C09078=1066.897,11.709,-66.020,172.395,25.660,154.694
C09079=1066.890,11.459,-66.005,172.394,25.657,154.694
C09080=1066.884,11.211,-65.991,172.393,25.655,154.694
C09081=1066.878,10.961,-65.976,172.391,25.653,154.693
C09082=1066.872,10.712,-65.961,172.390,25.650,154.693
C09083=1066.866,10.462,-65.946,172.388,25.647,154.693
C09084=1066.860,10.213,-65.931,172.387,25.645,154.692
C09085=1066.854,9.963,-65.918,172.386,25.642,154.692
C09086=1066.848,9.713,-65.903,172.384,25.640,154.692
C09087=1066.841,9.464,-65.888,172.383,25.637,154.692
C09088=1066.835,9.215,-65.873,172.381,25.635,154.691
C09089=1066.829,8.965,-65.858,172.380,25.632,154.691
C09090=1066.823,8.716,-65.844,172.378,25.630,154.691
C09091=1066.817,8.466,-65.829,172.377,25.627,154.690
C09092=1066.812,8.216,-65.814,172.376,25.625,154.690
C09093=1066.806,7.967,-65.799,172.374,25.622,154.690
C09094=1066.799,7.717,-65.784,172.373,25.619,154.689
C09095=1066.794,7.468,-65.770,172.371,25.617,154.689
C09096=1066.788,7.218,-65.755,172.370,25.615,154.689
C09097=1066.782,6.969,-65.741,172.369,25.612,154.688
C09098=1066.775,6.719,-65.726,172.367,25.610,154.688
C09099=1066.770,6.471,-65.711,172.366,25.607,154.688
C09100=1066.764,6.220,-65.697,172.364,25.604,154.687
C09101=1066.757,5.971,-65.682,172.363,25.602,154.687
C09102=1066.751,5.722,-65.668,172.361,25.600,154.687
C09103=1066.745,5.472,-65.653,172.360,25.597,154.686
C09104=1066.740,5.222,-65.639,172.359,25.594,154.686
C09105=1066.733,4.973,-65.624,172.357,25.592,154.686
C09106=1066.727,4.724,-65.609,172.356,25.589,154.686
C09107=1066.721,4.473,-65.595,172.354,25.587,154.685
C09108=1066.716,4.225,-65.580,172.353,25.584,154.685
C09109=1066.709,3.975,-65.565,172.352,25.582,154.685
C09110=1066.704,3.725,-65.552,172.350,25.579,154.684
C09111=1066.697,3.476,-65.537,172.349,25.577,154.684
C09112=1066.691,3.227,-65.522,172.347,25.574,154.684
C09113=1066.685,2.976,-65.508,172.346,25.572,154.683
C09114=1066.680,2.727,-65.493,172.344,25.569,154.683
C09115=1066.673,2.478,-65.478,172.343,25.566,154.683
C09116=1066.668,2.228,-65.464,172.342,25.564,154.682
C09117=1066.661,1.979,-65.450,172.340,25.562,154.682
C09118=1066.656,1.729,-65.436,172.339,25.559,154.682
C09119=1066.650,1.480,-65.421,172.337,25.556,154.681
C09120=1066.644,1.230,-65.406,172.336,25.554,154.681
C09121=1066.638,0.981,-65.392,172.334,25.551,154.681
C09122=1066.632,0.731,-65.377,172.333,25.549,154.681
C09123=1066.626,0.482,-65.363,172.332,25.547,154.680
C09124=1066.620,0.232,-65.348,172.330,25.544,154.680
C09125=1066.614,-0.017,-65.334,172.329,25.541,154.680
C09126=1066.608,-0.266,-65.321,172.327,25.539,154.679
C09127=1066.602,-0.516,-65.306,172.326,25.536,154.679
C09128=1066.596,-0.766,-65.292,172.325,25.534,154.679
C09129=1066.590,-1.015,-65.277,172.323,25.531,154.678
C09130=1066.584,-1.265,-65.263,172.322,25.528,154.678
C09131=1066.578,-1.545,-65.247,172.320,25.526,154.678
C09132=1066.571,-1.824,-65.231,172.319,25.523,154.677
C09133=1066.564,-2.105,-65.214,172.318,25.520,154.677
C09134=1066.557,-2.385,-65.198,172.315,25.517,154.677
C09135=1066.552,-2.634,-65.184,172.314,25.515,154.676
C09136=1066.546,-2.884,-65.171,172.312,25.512,154.676
C09137=1066.540,-3.133,-65.156,172.311,25.509,154.676
C09138=1066.534,-3.383,-65.142,172.310,25.507,154.675
C09139=1066.528,-3.633,-65.127,172.308,25.505,154.675
C09140=1066.522,-3.882,-65.114,172.307,25.502,154.675
C09141=1066.515,-4.132,-65.099,172.305,25.500,154.675
C09142=1066.510,-4.381,-65.085,172.304,25.498,154.674
C09143=1066.504,-4.631,-65.071,172.303,25.495,154.674
C09144=1066.497,-4.880,-65.057,172.301,25.493,154.674
C09145=1066.492,-5.130,-65.043,172.300,25.490,154.673
C09146=1066.485,-5.379,-65.028,172.298,25.488,154.673
C09147=1066.479,-5.629,-65.014,172.297,25.485,154.673
C09148=1066.473,-5.879,-65.000,172.295,25.483,154.673
C09149=1066.467,-6.128,-64.986,172.294,25.480,154.672
C09150=1066.461,-6.377,-64.972,172.293,25.478,154.672
C09151=1066.455,-6.627,-64.958,172.291,25.476,154.672
C09152=1066.449,-6.876,-64.944,172.290,25.473,154.671
C09153=1066.443,-7.125,-64.930,172.288,25.471,154.671
C09154=1066.437,-7.376,-64.916,172.287,25.469,154.671
C09155=1066.430,-7.624,-64.902,172.285,25.466,154.671
C09156=1066.424,-7.875,-64.888,172.284,25.463,154.670
C09157=1066.419,-8.124,-64.874,172.282,25.461,154.670
C09158=1066.412,-8.373,-64.860,172.281,25.459,154.670
C09159=1066.406,-8.623,-64.846,172.280,25.456,154.669
C09160=1066.401,-8.873,-64.832,172.278,25.454,154.669
C09161=1066.395,-9.122,-64.819,172.277,25.452,154.669
C09162=1066.388,-9.372,-64.804,172.275,25.449,154.669
C09163=1066.383,-9.621,-64.790,172.274,25.447,154.668
C09164=1066.377,-9.871,-64.777,172.272,25.444,154.668
C09165=1066.370,-10.121,-64.762,172.271,25.442,154.668
C09166=1066.364,-10.369,-64.748,172.270,25.439,154.667
C09167=1066.358,-10.619,-64.734,172.268,25.437,154.667
C09168=1066.352,-10.869,-64.720,172.267,25.435,154.667
C09169=1066.346,-11.119,-64.707,172.265,25.432,154.667
C09170=1066.341,-11.368,-64.693,172.264,25.430,154.666
C09171=1066.334,-11.617,-64.679,172.262,25.428,154.666
C09172=1066.328,-11.867,-64.665,172.261,25.425,154.666
C09173=1066.323,-12.117,-64.651,172.260,25.422,154.665
C09174=1066.316,-12.366,-64.638,172.258,25.420,154.665
C09175=1066.310,-12.616,-64.624,172.257,25.418,154.665
C09176=1066.304,-12.865,-64.610,172.255,25.415,154.664
C09177=1066.299,-13.115,-64.596,172.254,25.413,154.664
C09178=1066.292,-13.365,-64.581,172.252,25.411,154.664
C09179=1066.286,-13.614,-64.568,172.251,25.408,154.664
C09180=1066.281,-13.864,-64.554,172.249,25.405,154.663
C09181=1066.274,-14.113,-64.541,172.248,25.403,154.663
C09182=1066.268,-14.363,-64.527,172.247,25.401,154.663
C09183=1066.263,-14.613,-64.513,172.245,25.398,154.662
C09184=1066.257,-14.862,-64.500,172.244,25.396,154.662
C09185=1066.251,-15.111,-64.486,172.242,25.394,154.662
C09186=1066.244,-15.361,-64.472,172.241,25.391,154.662
C09187=1066.238,-15.611,-64.459,172.239,25.389,154.661
C09188=1066.233,-15.860,-64.445,172.238,25.386,154.661
C09189=1066.226,-16.109,-64.431,172.236,25.384,154.661
C09190=1066.220,-16.359,-64.417,172.235,25.382,154.661
C09191=1066.214,-16.608,-64.404,172.234,25.379,154.660
C09192=1066.208,-16.858,-64.390,172.232,25.377,154.660
C09193=1066.202,-17.108,-64.376,172.231,25.375,154.660
C09194=1066.195,-17.357,-64.363,172.229,25.372,154.660
C09195=1066.189,-17.636,-64.348,172.228,25.370,154.659
C09196=1066.182,-17.914,-64.333,172.225,25.367,154.659
C09197=1066.176,-18.193,-64.318,172.224,25.364,154.659
C09198=1066.169,-18.471,-64.302,172.223,25.362,154.658
C09199=1066.162,-18.720,-64.289,172.221,25.360,154.658
C09200=1066.156,-18.970,-64.276,172.220,25.357,154.658
C09201=1066.151,-19.220,-64.262,172.218,25.355,154.658
C09202=1066.144,-19.470,-64.249,172.217,25.353,154.657
C09203=1066.138,-19.719,-64.235,172.215,25.350,154.657
C09204=1066.132,-19.968,-64.221,172.214,25.348,154.657
C09205=1066.126,-20.218,-64.208,172.213,25.346,154.656
C09206=1066.119,-20.468,-64.195,172.211,25.343,154.656
C09207=1066.114,-20.717,-64.181,172.210,25.341,154.656
C09208=1066.108,-20.966,-64.167,172.208,25.339,154.656
C09209=1066.101,-21.216,-64.154,172.207,25.337,154.656
C09210=1066.096,-21.465,-64.140,172.205,25.334,154.655
C09211=1066.090,-21.715,-64.128,172.204,25.332,154.655
C09212=1066.083,-21.965,-64.114,172.202,25.330,154.655
C09213=1066.078,-22.215,-64.100,172.201,25.327,154.654
C09214=1066.072,-22.464,-64.087,172.199,25.325,154.654
C09215=1066.065,-22.713,-64.074,172.198,25.323,154.654
C09216=1066.060,-22.963,-64.060,172.197,25.320,154.654
C09217=1066.054,-23.212,-64.047,172.195,25.318,154.653
C09218=1066.047,-23.463,-64.034,172.194,25.316,154.653
C09219=1066.042,-23.712,-64.020,172.192,25.313,154.653
C09220=1066.035,-23.962,-64.007,172.191,25.311,154.653
C09221=1066.029,-24.211,-63.993,172.189,25.309,154.652
C09222=1066.024,-24.460,-63.979,172.187,25.306,154.652
C09223=1066.018,-24.710,-63.967,172.185,25.304,154.652
C09224=1066.012,-24.960,-63.954,172.184,25.302,154.652
C09225=1066.005,-25.209,-63.940,172.182,25.299,154.651
C09226=1066.000,-25.458,-63.926,172.181,25.297,154.651
C09227=1065.993,-25.709,-63.914,172.180,25.295,154.651
C09228=1065.987,-25.958,-63.900,172.178,25.292,154.651
C09229=1065.982,-26.208,-63.886,172.177,25.290,154.650
C09230=1065.976,-26.457,-63.873,172.175,25.288,154.650
C09231=1065.970,-26.707,-63.861,172.174,25.285,154.650
C09232=1065.963,-26.956,-63.847,172.172,25.283,154.650
C09233=1065.957,-27.205,-63.834,172.171,25.281,154.649
C09234=1065.951,-27.455,-63.821,172.169,25.279,154.649
C09235=1065.946,-27.705,-63.808,172.168,25.276,154.649
C09236=1065.939,-27.955,-63.794,172.166,25.274,154.649
C09237=1065.933,-28.205,-63.781,172.165,25.272,154.648
C09238=1065.927,-28.454,-63.768,172.163,25.270,154.648
C09239=1065.921,-28.703,-63.755,172.162,25.267,154.648
C09240=1065.915,-28.953,-63.742,172.161,25.265,154.648
C09241=1065.909,-29.202,-63.729,172.159,25.263,154.647
C09242=1065.902,-29.452,-63.716,172.158,25.261,154.647
C09243=1065.896,-29.702,-63.703,172.156,25.259,154.647
C09244=1065.890,-29.951,-63.690,172.155,25.256,154.647
C09245=1065.884,-30.201,-63.677,172.153,25.254,154.646
C09246=1065.878,-30.451,-63.664,172.152,25.252,154.646
C09247=1065.871,-30.700,-63.650,172.150,25.250,154.646
C09248=1065.865,-30.950,-63.638,172.149,25.247,154.646
C09249=1065.859,-31.199,-63.625,172.147,25.246,154.646
C09250=1065.854,-31.449,-63.612,172.146,25.243,154.645
C09251=1065.848,-31.699,-63.598,172.144,25.241,154.645
C09252=1065.842,-31.948,-63.586,172.143,25.239,154.645
C09253=1065.836,-32.198,-63.572,172.141,25.237,154.645
C09254=1065.829,-32.447,-63.559,172.140,25.234,154.644
C09255=1065.824,-32.697,-63.547,172.138,25.232,154.644
C09256=1065.817,-32.946,-63.533,172.137,25.230,154.644
C09257=1065.811,-33.196,-63.521,172.135,25.228,154.644
C09258=1065.805,-33.445,-63.508,172.134,25.226,154.643
C09259=1065.798,-33.723,-63.493,172.132,25.223,154.643
C09260=1065.791,-34.001,-63.479,172.130,25.220,154.643
C09261=1065.785,-34.279,-63.464,172.129,25.218,154.643
C09262=1065.778,-34.556,-63.450,172.127,25.216,154.642
C09263=1065.772,-34.806,-63.437,172.125,25.213,154.642
C09264=1065.766,-35.056,-63.424,172.123,25.211,154.642
C09265=1065.760,-35.305,-63.411,172.122,25.209,154.642
C09266=1065.754,-35.555,-63.399,172.121,25.207,154.641
C09267=1065.748,-35.805,-63.386,172.119,25.205,154.641
C09268=1065.742,-36.054,-63.373,172.118,25.202,154.641
C09269=1065.737,-36.303,-63.361,172.116,25.200,154.641
C09270=1065.730,-36.552,-63.347,172.115,25.198,154.641
C09271=1065.724,-36.802,-63.335,172.113,25.196,154.640
C09272=1065.718,-37.051,-63.322,172.112,25.194,154.640
C09273=1065.712,-37.301,-63.309,172.110,25.192,154.640
C09274=1065.706,-37.551,-63.296,172.109,25.189,154.640
C09275=1065.700,-37.801,-63.283,172.107,25.187,154.639
C09276=1065.694,-38.050,-63.271,172.106,25.185,154.639
C09277=1065.688,-38.300,-63.258,172.104,25.183,154.639
C09278=1065.682,-38.550,-63.245,172.103,25.181,154.639
C09279=1065.676,-38.799,-63.233,172.101,25.179,154.639
C09280=1065.670,-39.049,-63.220,172.100,25.176,154.638
C09281=1065.663,-39.298,-63.207,172.098,25.175,154.638
C09282=1065.658,-39.548,-63.194,172.097,25.172,154.638
C09283=1065.652,-39.798,-63.182,172.095,25.170,154.638
C09284=1065.645,-40.047,-63.169,172.094,25.168,154.637
C09285=1065.639,-40.297,-63.157,172.092,25.166,154.637
C09286=1065.633,-40.547,-63.144,172.091,25.164,154.637
C09287=1065.627,-40.796,-63.131,172.089,25.162,154.637
C09288=1065.621,-41.046,-63.118,172.088,25.160,154.637
C09289=1065.614,-41.295,-63.106,172.086,25.158,154.637
C09290=1065.609,-41.545,-63.094,172.085,25.156,154.636
C09291=1065.603,-41.794,-63.081,172.083,25.154,154.636
C09292=1065.597,-42.044,-63.068,172.081,25.151,154.636
C09293=1065.590,-42.293,-63.056,172.079,25.149,154.636
C09294=1065.584,-42.543,-63.044,172.078,25.147,154.635
C09295=1065.578,-42.793,-63.031,172.076,25.145,154.635
C09296=1065.572,-43.042,-63.018,172.075,25.143,154.635
C09297=1065.565,-43.292,-63.006,172.073,25.141,154.635
C09298=1065.559,-43.542,-62.993,172.072,25.139,154.635
C09299=1065.554,-43.792,-62.981,172.070,25.137,154.635
C09300=1065.548,-44.042,-62.968,172.069,25.134,154.634
C09301=1065.541,-44.290,-62.956,172.067,25.133,154.634
C09302=1065.535,-44.540,-62.943,172.066,25.130,154.634
C09303=1065.529,-44.790,-62.931,172.064,25.128,154.634
C09304=1065.524,-45.040,-62.918,172.063,25.126,154.633
C09305=1065.517,-45.289,-62.906,172.061,25.124,154.633
C09306=1065.511,-45.539,-62.894,172.060,25.122,154.633
C09307=1065.505,-45.789,-62.881,172.058,25.120,154.633
C09308=1065.499,-46.037,-62.869,172.057,25.118,154.633
C09309=1065.493,-46.287,-62.856,172.055,25.116,154.632
C09310=1065.487,-46.537,-62.844,172.054,25.114,154.632
C09311=1065.481,-46.787,-62.831,172.052,25.112,154.632
C09312=1065.474,-47.036,-62.819,172.051,25.110,154.632
C09313=1065.468,-47.286,-62.807,172.049,25.108,154.632
C09314=1065.463,-47.535,-62.795,172.048,25.106,154.631
C09315=1065.456,-47.785,-62.783,172.046,25.103,154.631
C09316=1065.451,-48.035,-62.770,172.045,25.102,154.631
C09317=1065.445,-48.285,-62.758,172.043,25.100,154.631
C09318=1065.439,-48.535,-62.745,172.041,25.097,154.631
C09319=1065.433,-48.783,-62.733,172.039,25.095,154.631
C09320=1065.427,-49.033,-62.721,172.038,25.093,154.630
C09321=1065.421,-49.283,-62.708,172.036,25.091,154.630
C09322=1065.414,-49.533,-62.696,172.035,25.089,154.630
C09323=1065.407,-49.811,-62.682,172.033,25.087,154.630
C09324=1065.401,-50.089,-62.669,172.032,25.085,154.629
C09325=1065.394,-50.366,-62.655,172.029,25.083,154.629
C09326=1065.388,-50.644,-62.641,172.028,25.080,154.629
C09327=1065.381,-50.894,-62.630,172.026,25.078,154.629
C09328=1065.375,-51.144,-62.617,172.025,25.077,154.629
C09329=1065.369,-51.393,-62.605,172.023,25.074,154.629
C09330=1065.362,-51.643,-62.593,172.022,25.072,154.628
C09331=1065.356,-51.893,-62.580,172.020,25.071,154.628
C09332=1065.349,-52.142,-62.569,172.019,25.069,154.628
C09333=1065.344,-52.391,-62.556,172.017,25.067,154.628
C09334=1065.338,-52.642,-62.545,172.016,25.065,154.628
C09335=1065.331,-52.891,-62.533,172.014,25.063,154.628
C09336=1065.325,-53.141,-62.521,172.013,25.061,154.627
C09337=1065.319,-53.391,-62.509,172.011,25.059,154.627
C09338=1065.313,-53.640,-62.496,172.009,25.057,154.627
C09339=1065.307,-53.889,-62.484,172.008,25.056,154.627
C09340=1065.300,-54.139,-62.473,172.006,25.054,154.627
C09341=1065.294,-54.389,-62.460,172.005,25.052,154.627
C09342=1065.288,-54.639,-62.449,172.002,25.049,154.627
C09343=1065.282,-54.888,-62.437,172.001,25.048,154.626
C09344=1065.276,-55.138,-62.425,171.999,25.046,154.626
C09345=1065.269,-55.387,-62.413,171.998,25.044,154.626
C09346=1065.263,-55.637,-62.400,171.996,25.042,154.626
C09347=1065.257,-55.886,-62.388,171.995,25.040,154.626
C09348=1065.251,-56.136,-62.377,171.993,25.038,154.626
C09349=1065.245,-56.386,-62.365,171.992,25.036,154.625
C09350=1065.238,-56.636,-62.353,171.990,25.034,154.625
C09351=1065.232,-56.885,-62.341,171.988,25.033,154.625
C09352=1065.226,-57.135,-62.329,171.987,25.031,154.625
C09353=1065.220,-57.385,-62.317,171.985,25.029,154.625
C09354=1065.213,-57.634,-62.305,171.984,25.027,154.625
C09355=1065.208,-57.884,-62.293,171.982,25.025,154.625
C09356=1065.201,-58.133,-62.281,171.981,25.023,154.624
C09357=1065.195,-58.383,-62.270,171.979,25.021,154.624
C09358=1065.189,-58.633,-62.257,171.978,25.019,154.624
C09359=1065.183,-58.882,-62.246,171.976,25.018,154.624
C09360=1065.177,-59.132,-62.235,171.975,25.016,154.624
C09361=1065.171,-59.382,-62.222,171.973,25.014,154.624
C09362=1065.165,-59.631,-62.210,171.971,25.012,154.623
C09363=1065.158,-59.881,-62.199,171.969,25.010,154.623
C09364=1065.153,-60.131,-62.187,171.967,25.008,154.623
C09365=1065.146,-60.380,-62.175,171.966,25.006,154.623
C09366=1065.140,-60.629,-62.163,171.964,25.005,154.623
C09367=1065.134,-60.880,-62.151,171.963,25.003,154.623
C09368=1065.128,-61.129,-62.140,171.961,25.001,154.622
C09369=1065.122,-61.379,-62.128,171.960,24.999,154.622
C09370=1065.116,-61.629,-62.116,171.958,24.997,154.622
C09371=1065.110,-61.878,-62.104,171.957,24.995,154.622
C09372=1065.104,-62.128,-62.093,171.955,24.993,154.622
C09373=1065.097,-62.378,-62.081,171.953,24.991,154.622
C09374=1065.092,-62.627,-62.069,171.952,24.990,154.622
C09375=1065.085,-62.877,-62.058,171.950,24.988,154.621
C09376=1065.079,-63.126,-62.046,171.949,24.986,154.621
C09377=1065.074,-63.376,-62.034,171.947,24.984,154.621
C09378=1065.067,-63.626,-62.022,171.946,24.982,154.621
C09379=1065.061,-63.875,-62.011,171.944,24.981,154.621
C09380=1065.055,-64.125,-61.999,171.942,24.979,154.621
C09381=1065.049,-64.375,-61.987,171.941,24.977,154.621
C09382=1065.043,-64.624,-61.976,171.939,24.975,154.620
C09383=1065.036,-64.874,-61.964,171.938,24.973,154.620
C09384=1065.031,-65.123,-61.953,171.935,24.971,154.620
C09385=1065.025,-65.373,-61.941,171.934,24.970,154.620
C09386=1065.019,-65.623,-61.930,171.932,24.968,154.620
C09387=1065.012,-65.902,-61.917,171.931,24.966,154.620
C09388=1065.005,-66.182,-61.904,171.929,24.964,154.620
C09389=1064.998,-66.460,-61.890,171.928,24.962,154.620
C09390=1064.992,-66.740,-61.877,171.925,24.960,154.619
C09391=1064.986,-66.990,-61.866,171.924,24.958,154.619
C09392=1064.979,-67.239,-61.854,171.922,24.956,154.619
C09393=1064.973,-67.489,-61.843,171.920,24.955,154.619
C09394=1064.967,-67.738,-61.831,171.919,24.953,154.619
C09395=1064.961,-67.989,-61.819,171.917,24.951,154.619
C09396=1064.955,-68.238,-61.809,171.916,24.949,154.619
C09397=1064.949,-68.488,-61.797,171.914,24.948,154.618
C09398=1064.943,-68.737,-61.786,171.913,24.946,154.618
C09399=1064.937,-68.987,-61.773,171.911,24.944,154.618
C09400=1064.931,-69.237,-61.762,171.909,24.942,154.618
C09401=1064.925,-69.487,-61.751,171.908,24.940,154.618
C09402=1064.919,-69.736,-61.739,171.906,24.938,154.618
C09403=1064.913,-69.986,-61.728,171.905,24.937,154.618
C09404=1064.907,-70.235,-61.716,171.903,24.935,154.617
C09405=1064.901,-70.485,-61.705,171.902,24.933,154.617
C09406=1064.895,-70.735,-61.694,171.899,24.932,154.617
C09407=1064.889,-70.984,-61.682,171.897,24.930,154.617
C09408=1064.883,-71.234,-61.671,171.896,24.928,154.617
C09409=1064.877,-71.484,-61.659,171.894,24.926,154.617
C09410=1064.871,-71.733,-61.648,171.893,24.924,154.617
C09411=1064.866,-71.983,-61.637,171.891,24.922,154.617
C09412=1064.859,-72.233,-61.626,171.890,24.921,154.616
C09413=1064.853,-72.482,-61.614,171.888,24.919,154.616
C09414=1064.848,-72.732,-61.602,171.886,24.918,154.616
C09415=1064.842,-72.982,-61.591,171.885,24.916,154.616
C09416=1064.835,-73.231,-61.579,171.883,24.914,154.616
C09417=1064.829,-73.481,-61.568,171.882,24.912,154.616
C09418=1064.823,-73.731,-61.557,171.880,24.910,154.616
C09419=1064.817,-73.981,-61.546,171.879,24.909,154.616
C09420=1064.811,-74.229,-61.535,171.877,24.907,154.616
C09421=1064.805,-74.480,-61.523,171.875,24.906,154.615
C09422=1064.799,-74.729,-61.513,171.874,24.904,154.615
C09423=1064.793,-74.979,-61.501,171.872,24.903,154.615
C09424=1064.787,-75.228,-61.490,171.871,24.901,154.615
C09425=1064.781,-75.478,-61.478,171.869,24.899,154.615
C09426=1064.775,-75.728,-61.468,171.867,24.898,154.615
C09427=1064.768,-75.978,-61.456,171.866,24.896,154.615
C09428=1064.763,-76.228,-61.445,171.863,24.894,154.615
C09429=1064.756,-76.477,-61.434,171.862,24.892,154.615
C09430=1064.750,-76.727,-61.423,171.860,24.891,154.615
C09431=1064.744,-76.977,-61.411,171.858,24.889,154.614
C09432=1064.738,-77.226,-61.401,171.857,24.888,154.614
C09433=1064.732,-77.476,-61.390,171.855,24.886,154.614
C09434=1064.726,-77.726,-61.378,171.854,24.884,154.614
C09435=1064.720,-77.975,-61.367,171.852,24.883,154.614
C09436=1064.714,-78.225,-61.356,171.850,24.881,154.614
C09437=1064.707,-78.474,-61.345,171.849,24.880,154.614
C09438=1064.702,-78.724,-61.334,171.847,24.878,154.614
C09439=1064.695,-78.974,-61.323,171.846,24.876,154.614
C09440=1064.689,-79.223,-61.312,171.844,24.875,154.614
C09441=1064.683,-79.474,-61.301,171.842,24.873,154.614
C09442=1064.677,-79.723,-61.290,171.841,24.872,154.614
C09443=1064.672,-79.973,-61.279,171.839,24.870,154.613
C09444=1064.665,-80.223,-61.268,171.837,24.869,154.613
C09445=1064.659,-80.471,-61.257,171.836,24.867,154.613
C09446=1064.652,-80.721,-61.246,171.834,24.866,154.613
C09447=1064.646,-80.971,-61.235,171.833,24.864,154.613
C09448=1064.639,-81.221,-61.224,171.831,24.863,154.613
C09449=1064.634,-81.470,-61.213,171.828,24.861,154.613
C09450=1064.628,-81.720,-61.203,171.827,24.859,154.613
C09451=1064.620,-82.002,-61.190,171.825,24.858,154.613
C09452=1064.614,-82.284,-61.178,171.823,24.856,154.613
C09453=1064.606,-82.565,-61.165,171.822,24.854,154.613
C09454=1064.599,-82.846,-61.153,171.819,24.852,154.613
C09455=1064.594,-83.096,-61.142,171.818,24.851,154.613
C09456=1064.587,-83.345,-61.132,171.816,24.850,154.613
C09457=1064.581,-83.595,-61.121,171.814,24.848,154.612
C09458=1064.575,-83.845,-61.110,171.813,24.847,154.612
C09459=1064.569,-84.094,-61.100,171.811,24.845,154.612
C09460=1064.562,-84.344,-61.088,171.810,24.844,154.612
C09461=1064.557,-84.594,-61.078,171.808,24.843,154.612
C09462=1064.550,-84.844,-61.068,171.806,24.841,154.612
C09463=1064.544,-85.094,-61.057,171.805,24.839,154.612
C09464=1064.538,-85.343,-61.046,171.803,24.838,154.612
C09465=1064.531,-85.593,-61.035,171.801,24.836,154.612
C09466=1064.526,-85.843,-61.024,171.800,24.835,154.612
C09467=1064.520,-86.092,-61.014,171.798,24.833,154.612
C09468=1064.513,-86.342,-61.003,171.796,24.832,154.612
C09469=1064.507,-86.591,-60.992,171.795,24.831,154.612
C09470=1064.501,-86.841,-60.981,171.792,24.829,154.612
C09471=1064.494,-87.091,-60.970,171.790,24.828,154.612
C09472=1064.489,-87.341,-60.960,171.789,24.826,154.612
C09473=1064.483,-87.590,-60.949,171.787,24.824,154.611
C09474=1064.476,-87.840,-60.939,171.786,24.823,154.611
C09475=1064.470,-88.090,-60.928,171.784,24.822,154.611
C09476=1064.464,-88.339,-60.917,171.782,24.821,154.611
C09477=1064.458,-88.588,-60.907,171.781,24.819,154.611
C09478=1064.452,-88.839,-60.896,171.779,24.818,154.611
C09479=1064.446,-89.089,-60.885,171.777,24.816,154.611
C09480=1064.440,-89.338,-60.875,171.776,24.815,154.611
C09481=1064.434,-89.587,-60.864,171.774,24.813,154.611
C09482=1064.427,-89.837,-60.854,171.772,24.812,154.611
C09483=1064.421,-90.087,-60.843,171.771,24.811,154.611
C09484=1064.416,-90.337,-60.832,171.769,24.809,154.611
C09485=1064.409,-90.587,-60.822,171.767,24.808,154.611
C09486=1064.403,-90.836,-60.811,171.766,24.807,154.611
C09487=1064.397,-91.086,-60.801,171.764,24.805,154.611
C09488=1064.391,-91.335,-60.791,171.762,24.804,154.611
C09489=1064.385,-91.585,-60.780,171.761,24.802,154.611
C09490=1064.378,-91.835,-60.769,171.759,24.801,154.611
C09491=1064.373,-92.085,-60.759,171.757,24.800,154.611
C09492=1064.367,-92.334,-60.748,171.756,24.798,154.610
C09493=1064.361,-92.584,-60.738,171.754,24.797,154.610
C09494=1064.354,-92.834,-60.727,171.751,24.795,154.611
C09495=1064.348,-93.084,-60.717,171.750,24.794,154.610
C09496=1064.342,-93.333,-60.706,171.748,24.793,154.610
C09497=1064.337,-93.583,-60.696,171.746,24.791,154.610
C09498=1064.330,-93.832,-60.686,171.745,24.790,154.610
C09499=1064.324,-94.083,-60.674,171.743,24.789,154.610
C09500=1064.318,-94.332,-60.665,171.741,24.787,154.610
C09501=1064.312,-94.582,-60.654,171.740,24.786,154.610
C09502=1064.306,-94.831,-60.643,171.738,24.784,154.610
C09503=1064.300,-95.081,-60.633,171.736,24.783,154.610
C09504=1064.294,-95.331,-60.623,171.735,24.782,154.610
C09505=1064.288,-95.581,-60.613,171.733,24.781,154.610
C09506=1064.282,-95.831,-60.602,171.731,24.779,154.610
C09507=1064.275,-96.080,-60.591,171.730,24.778,154.610
C09508=1064.270,-96.330,-60.581,171.728,24.777,154.610
C09509=1064.264,-96.579,-60.571,171.726,24.775,154.610
C09510=1064.258,-96.829,-60.561,171.725,24.774,154.610
C09511=1064.252,-97.079,-60.550,171.723,24.773,154.610
C09512=1064.245,-97.329,-60.539,171.721,24.771,154.610
C09513=1064.240,-97.579,-60.529,171.720,24.770,154.610
C09514=1064.233,-97.828,-60.519,171.718,24.769,154.610
C09515=1064.227,-98.112,-60.508,171.715,24.767,154.610
C09516=1064.220,-98.396,-60.496,171.714,24.766,154.610
C09517=1064.213,-98.679,-60.484,171.712,24.765,154.610
C09518=1064.205,-98.963,-60.473,171.710,24.763,154.610
C09519=1064.199,-99.213,-60.462,171.708,24.762,154.610
C09520=1064.193,-99.463,-60.452,171.706,24.761,154.610
C09521=1064.187,-99.712,-60.442,171.704,24.759,154.610
C09522=1064.181,-99.962,-60.432,171.703,24.758,154.610
C09523=1064.175,-100.211,-60.422,171.701,24.757,154.610
C09524=1064.168,-100.462,-60.412,171.699,24.756,154.610
C09525=1064.162,-100.711,-60.401,171.697,24.754,154.610
C09526=1064.156,-100.961,-60.391,171.696,24.753,154.610
C09527=1064.150,-101.210,-60.381,171.694,24.752,154.610
C09528=1064.144,-101.460,-60.371,171.692,24.751,154.610
C09529=1064.138,-101.710,-60.361,171.691,24.750,154.610
C09530=1064.132,-101.959,-60.351,171.689,24.749,154.610
C09531=1064.126,-102.209,-60.341,171.687,24.748,154.610
C09532=1064.120,-102.459,-60.331,171.685,24.746,154.610
C09533=1064.113,-102.709,-60.321,171.684,24.745,154.610
C09534=1064.107,-102.959,-60.311,171.682,24.744,154.610
C09535=1064.101,-103.208,-60.300,171.680,24.743,154.610
C09536=1064.095,-103.458,-60.291,171.679,24.741,154.610
C09537=1064.089,-103.708,-60.280,171.677,24.741,154.610
C09538=1064.083,-103.957,-60.270,171.675,24.740,154.610
C09539=1064.077,-104.207,-60.261,171.673,24.738,154.610
C09540=1064.070,-104.456,-60.250,171.672,24.737,154.610
C09541=1064.065,-104.707,-60.240,171.670,24.736,154.610
C09542=1064.059,-104.956,-60.231,171.668,24.735,154.610
C09543=1064.052,-105.205,-60.220,171.667,24.734,154.610
C09544=1064.046,-105.455,-60.211,171.665,24.733,154.610
C09545=1064.041,-105.705,-60.201,171.663,24.731,154.610
C09546=1064.034,-105.955,-60.190,171.661,24.730,154.610
C09547=1064.027,-106.205,-60.180,171.660,24.729,154.610
C09548=1064.021,-106.455,-60.171,171.658,24.728,154.610
C09549=1064.016,-106.705,-60.161,171.656,24.727,154.610
C09550=1064.009,-106.954,-60.150,171.655,24.726,154.610
C09551=1064.003,-107.204,-60.141,171.653,24.725,154.610
C09552=1063.997,-107.454,-60.131,171.651,24.724,154.610
C09553=1063.991,-107.704,-60.122,171.649,24.723,154.610
C09554=1063.985,-107.953,-60.111,171.647,24.721,154.610
C09555=1063.979,-108.203,-60.101,171.645,24.720,154.610
C09556=1063.973,-108.453,-60.092,171.643,24.719,154.610
C09557=1063.966,-108.702,-60.082,171.641,24.718,154.610
C09558=1063.960,-108.952,-60.072,171.640,24.717,154.610
C09559=1063.954,-109.201,-60.062,171.638,24.716,154.610
C09560=1063.948,-109.451,-60.053,171.636,24.715,154.610
C09561=1063.941,-109.701,-60.043,171.634,24.714,154.610
C09562=1063.936,-109.951,-60.033,171.633,24.713,154.610
C09563=1063.930,-110.200,-60.023,171.631,24.712,154.610
C09564=1063.923,-110.450,-60.013,171.629,24.711,154.610
C09565=1063.917,-110.700,-60.004,171.627,24.710,154.610
C09566=1063.911,-110.950,-59.994,171.626,24.709,154.610
C09567=1063.905,-111.199,-59.984,171.624,24.708,154.610
C09568=1063.899,-111.449,-59.975,171.622,24.707,154.610
C09569=1063.893,-111.699,-59.965,171.620,24.706,154.610
C09570=1063.886,-111.948,-59.955,171.619,24.705,154.610
C09571=1063.880,-112.198,-59.945,171.617,24.704,154.611
C09572=1063.874,-112.448,-59.935,171.615,24.703,154.611
C09573=1063.868,-112.698,-59.926,171.613,24.702,154.611
C09574=1063.862,-112.948,-59.916,171.612,24.701,154.611
C09575=1063.856,-113.198,-59.907,171.610,24.700,154.611
C09576=1063.850,-113.447,-59.897,171.608,24.699,154.611
C09577=1063.844,-113.697,-59.887,171.606,24.698,154.611
C09578=1063.837,-113.947,-59.878,171.605,24.697,154.611
C09579=1063.830,-114.229,-59.867,171.603,24.696,154.611
C09580=1063.824,-114.510,-59.856,171.600,24.695,154.611
C09581=1063.817,-114.792,-59.845,171.598,24.694,154.611
C09582=1063.810,-115.074,-59.835,171.597,24.693,154.611
C09583=1063.803,-115.324,-59.825,171.595,24.692,154.611
C09584=1063.797,-115.574,-59.816,171.593,24.691,154.611
C09585=1063.791,-115.824,-59.806,171.591,24.690,154.611
C09586=1063.785,-116.074,-59.796,171.589,24.689,154.611
C09587=1063.779,-116.323,-59.787,171.588,24.688,154.611
C09588=1063.772,-116.573,-59.777,171.586,24.687,154.611
C09589=1063.766,-116.823,-59.768,171.584,24.687,154.611
C09590=1063.761,-117.072,-59.759,171.582,24.685,154.611
C09591=1063.755,-117.322,-59.749,171.581,24.685,154.612
C09592=1063.748,-117.572,-59.739,171.579,24.684,154.612
C09593=1063.742,-117.821,-59.730,171.577,24.683,154.612
C09594=1063.736,-118.071,-59.720,171.575,24.682,154.612
C09595=1063.730,-118.321,-59.711,171.573,24.681,154.612
C09596=1063.724,-118.571,-59.701,171.572,24.680,154.612
C09597=1063.718,-118.821,-59.692,171.570,24.680,154.612
C09598=1063.711,-119.070,-59.682,171.568,24.679,154.612
C09599=1063.704,-119.320,-59.673,171.566,24.678,154.612
C09600=1063.699,-119.569,-59.664,171.564,24.677,154.612
C09601=1063.693,-119.819,-59.655,171.563,24.676,154.612
C09602=1063.687,-120.069,-59.645,171.561,24.675,154.612
C09603=1063.681,-120.319,-59.636,171.559,24.674,154.612
C09604=1063.675,-120.569,-59.626,171.557,24.674,154.612
C09605=1063.668,-120.819,-59.617,171.556,24.673,154.612
C09606=1063.662,-121.068,-59.607,171.554,24.672,154.613
C09607=1063.656,-121.318,-59.598,171.552,24.671,154.613
C09608=1063.650,-121.568,-59.590,171.550,24.671,154.613
C09609=1063.644,-121.817,-59.580,171.548,24.669,154.613
C09610=1063.638,-122.067,-59.571,171.547,24.669,154.613
C09611=1063.631,-122.317,-59.561,171.545,24.668,154.613
C09612=1063.625,-122.567,-59.551,171.543,24.667,154.613
C09613=1063.619,-122.817,-59.542,171.541,24.666,154.613
C09614=1063.614,-123.066,-59.533,171.539,24.665,154.613
C09615=1063.607,-123.316,-59.524,171.537,24.665,154.613
C09616=1063.601,-123.566,-59.515,171.536,24.664,154.613
C09617=1063.595,-123.815,-59.505,171.534,24.663,154.613
C09618=1063.588,-124.065,-59.496,171.532,24.662,154.613
C09619=1063.583,-124.316,-59.487,171.530,24.662,154.614
C09620=1063.576,-124.564,-59.478,171.528,24.661,154.614
C09621=1063.570,-124.814,-59.469,171.527,24.660,154.614
C09622=1063.564,-125.064,-59.459,171.525,24.660,154.614
C09623=1063.558,-125.314,-59.450,171.523,24.659,154.614
C09624=1063.551,-125.564,-59.441,171.521,24.658,154.614
C09625=1063.546,-125.813,-59.432,171.519,24.658,154.614
C09626=1063.540,-126.063,-59.423,171.518,24.656,154.614
C09627=1063.534,-126.313,-59.414,171.516,24.656,154.614
C09628=1063.527,-126.563,-59.405,171.514,24.655,154.614
C09629=1063.520,-126.813,-59.395,171.512,24.654,154.615
C09630=1063.515,-127.062,-59.387,171.510,24.654,154.615
C09631=1063.508,-127.312,-59.378,171.508,24.653,154.615
C09632=1063.502,-127.562,-59.368,171.506,24.652,154.615
C09633=1063.496,-127.812,-59.359,171.505,24.652,154.615
C09634=1063.491,-128.061,-59.350,171.503,24.650,154.615
C09635=1063.487,-128.312,-59.339,171.501,24.649,154.615
C09636=1063.485,-128.563,-59.329,171.500,24.647,154.615
C09637=1063.484,-128.814,-59.316,171.499,24.644,154.614
C09638=1063.485,-129.064,-59.304,171.498,24.640,154.614
C09639=1063.488,-129.316,-59.290,171.497,24.636,154.613
C09640=1063.493,-129.567,-59.276,171.497,24.631,154.612
C09641=1063.498,-129.819,-59.262,171.496,24.626,154.611
C09642=1063.506,-130.069,-59.246,171.496,24.620,154.610
C09643=1063.123,-130.092,-59.431,171.448,24.772,154.643
C09644=1063.115,-129.842,-59.447,171.449,24.778,154.644
C09645=1063.110,-129.590,-59.461,171.448,24.784,154.645
C09646=1063.106,-129.339,-59.476,171.449,24.788,154.646
C09647=1063.103,-129.086,-59.490,171.450,24.792,154.647
C09648=1063.102,-128.836,-59.502,171.451,24.796,154.647
C09649=1063.102,-128.586,-59.514,171.453,24.799,154.648
C09650=1063.105,-128.335,-59.525,171.454,24.801,154.648
C09651=1063.108,-128.084,-59.535,171.456,24.803,154.648
C09652=1063.112,-127.835,-59.545,171.457,24.804,154.648
C09653=1063.119,-127.585,-59.553,171.459,24.805,154.648
C09654=1063.125,-127.335,-59.563,171.461,24.806,154.648
C09655=1063.131,-127.085,-59.572,171.463,24.806,154.648
C09656=1063.138,-126.835,-59.581,171.465,24.807,154.648
C09657=1063.144,-126.586,-59.590,171.466,24.808,154.647
C09658=1063.150,-126.336,-59.599,171.468,24.808,154.647
C09659=1063.156,-126.086,-59.609,171.470,24.809,154.647
C09660=1063.163,-125.836,-59.617,171.472,24.810,154.647
C09661=1063.169,-125.586,-59.627,171.474,24.810,154.647
C09662=1063.174,-125.337,-59.636,171.476,24.811,154.647
C09663=1063.180,-125.087,-59.645,171.478,24.812,154.647
C09664=1063.187,-124.837,-59.654,171.479,24.813,154.647
C09665=1063.193,-124.587,-59.663,171.481,24.814,154.647
C09666=1063.199,-124.338,-59.673,171.483,24.814,154.647
C09667=1063.205,-124.087,-59.682,171.485,24.815,154.646
C09668=1063.212,-123.838,-59.690,171.487,24.815,154.646
C09669=1063.218,-123.589,-59.700,171.488,24.816,154.646
C09670=1063.224,-123.339,-59.710,171.490,24.817,154.646
C09671=1063.230,-123.089,-59.719,171.492,24.818,154.646
C09672=1063.236,-122.839,-59.728,171.494,24.819,154.646
C09673=1063.242,-122.590,-59.737,171.496,24.819,154.646
C09674=1063.248,-122.340,-59.747,171.497,24.821,154.646
C09675=1063.255,-122.090,-59.756,171.499,24.821,154.646
C09676=1063.261,-121.840,-59.765,171.501,24.822,154.646
C09677=1063.267,-121.591,-59.775,171.503,24.823,154.646
C09678=1063.273,-121.340,-59.784,171.505,24.823,154.646
C09679=1063.279,-121.090,-59.793,171.506,24.824,154.646
C09680=1063.285,-120.841,-59.802,171.508,24.825,154.645
C09681=1063.291,-120.592,-59.812,171.510,24.826,154.645
C09682=1063.298,-120.342,-59.821,171.512,24.827,154.645
C09683=1063.304,-120.092,-59.831,171.514,24.828,154.645
C09684=1063.310,-119.842,-59.840,171.515,24.828,154.645
C09685=1063.316,-119.592,-59.849,171.517,24.829,154.645
C09686=1063.322,-119.342,-59.859,171.519,24.830,154.645
C09687=1063.328,-119.092,-59.868,171.521,24.831,154.645
C09688=1063.334,-118.843,-59.877,171.523,24.831,154.645
C09689=1063.340,-118.594,-59.887,171.524,24.833,154.645
C09690=1063.346,-118.344,-59.896,171.526,24.833,154.645
C09691=1063.352,-118.094,-59.906,171.528,24.835,154.645
C09692=1063.359,-117.844,-59.915,171.530,24.835,154.645
C09693=1063.365,-117.595,-59.925,171.532,24.836,154.645
C09694=1063.372,-117.345,-59.934,171.533,24.837,154.645
C09695=1063.378,-117.095,-59.944,171.535,24.838,154.644
C09696=1063.384,-116.845,-59.953,171.537,24.838,154.644
C09697=1063.390,-116.595,-59.963,171.539,24.840,154.644
C09698=1063.396,-116.346,-59.972,171.541,24.840,154.644
C09699=1063.402,-116.097,-59.982,171.542,24.842,154.644
C09700=1063.408,-115.847,-59.991,171.544,24.842,154.644
C09701=1063.414,-115.597,-60.001,171.546,24.843,154.644
C09702=1063.420,-115.347,-60.010,171.548,24.844,154.644
C09703=1063.426,-115.097,-60.020,171.549,24.845,154.644
C09704=1063.434,-114.815,-60.031,171.551,24.846,154.644
C09705=1063.440,-114.533,-60.042,171.554,24.847,154.644
C09706=1063.447,-114.251,-60.052,171.556,24.848,154.644
C09707=1063.454,-113.968,-60.063,171.557,24.849,154.644
C09708=1063.460,-113.719,-60.073,171.559,24.850,154.644
C09709=1063.467,-113.469,-60.083,171.561,24.851,154.644
C09710=1063.473,-113.220,-60.093,171.563,24.852,154.644
C09711=1063.479,-112.970,-60.102,171.564,24.853,154.644
C09712=1063.485,-112.720,-60.112,171.566,24.854,154.644
C09713=1063.491,-112.470,-60.121,171.568,24.855,154.644
C09714=1063.497,-112.220,-60.131,171.570,24.856,154.643
C09715=1063.503,-111.971,-60.140,171.572,24.857,154.643
C09716=1063.509,-111.721,-60.150,171.573,24.858,154.643
C09717=1063.515,-111.472,-60.159,171.575,24.859,154.643
C09718=1063.521,-111.222,-60.170,171.577,24.860,154.643
C09719=1063.527,-110.972,-60.180,171.579,24.861,154.643
C09720=1063.533,-110.723,-60.189,171.580,24.862,154.643
C09721=1063.540,-110.473,-60.199,171.583,24.863,154.643
C09722=1063.546,-110.223,-60.208,171.585,24.864,154.643
C09723=1063.552,-109.973,-60.218,171.586,24.865,154.643
C09724=1063.558,-109.724,-60.228,171.588,24.866,154.643
C09725=1063.565,-109.474,-60.238,171.590,24.867,154.643
C09726=1063.571,-109.224,-60.248,171.592,24.869,154.643
C09727=1063.577,-108.974,-60.258,171.594,24.869,154.643
C09728=1063.583,-108.724,-60.267,171.595,24.870,154.643
C09729=1063.589,-108.475,-60.278,171.597,24.871,154.643
C09730=1063.596,-108.225,-60.287,171.599,24.872,154.643
C09731=1063.602,-107.975,-60.297,171.600,24.874,154.643
C09732=1063.608,-107.725,-60.306,171.602,24.874,154.643
C09733=1063.614,-107.476,-60.317,171.604,24.875,154.643
C09734=1063.620,-107.226,-60.327,171.606,24.877,154.643
C09735=1063.626,-106.976,-60.336,171.607,24.878,154.643
C09736=1063.632,-106.726,-60.346,171.609,24.879,154.643
C09737=1063.639,-106.477,-60.356,171.611,24.880,154.643
C09738=1063.645,-106.227,-60.366,171.613,24.881,154.643
C09739=1063.650,-105.977,-60.376,171.614,24.882,154.643
C09740=1063.657,-105.728,-60.386,171.616,24.883,154.643
C09741=1063.663,-105.478,-60.396,171.618,24.884,154.643
C09742=1063.669,-105.228,-60.405,171.620,24.885,154.643
C09743=1063.675,-104.978,-60.416,171.621,24.887,154.643
C09744=1063.681,-104.729,-60.426,171.623,24.888,154.643
C09745=1063.687,-104.479,-60.435,171.625,24.888,154.643
C09746=1063.693,-104.229,-60.446,171.627,24.890,154.643
C09747=1063.700,-103.979,-60.456,171.628,24.891,154.643
C09748=1063.706,-103.730,-60.466,171.630,24.892,154.643
C09749=1063.712,-103.480,-60.476,171.632,24.893,154.643
C09750=1063.718,-103.230,-60.486,171.633,24.895,154.643
C09751=1063.724,-102.981,-60.496,171.635,24.895,154.643
C09752=1063.730,-102.731,-60.506,171.637,24.897,154.643
C09753=1063.736,-102.481,-60.516,171.639,24.898,154.643
C09754=1063.742,-102.232,-60.527,171.640,24.899,154.643
C09755=1063.749,-101.982,-60.536,171.643,24.901,154.643
C09756=1063.754,-101.732,-60.546,171.645,24.902,154.643
C09757=1063.761,-101.482,-60.557,171.646,24.903,154.643
C09758=1063.767,-101.232,-60.567,171.648,24.904,154.643
C09759=1063.773,-100.983,-60.577,171.650,24.905,154.643
C09760=1063.779,-100.733,-60.587,171.652,24.906,154.643
C09761=1063.786,-100.484,-60.597,171.653,24.907,154.643
C09762=1063.791,-100.234,-60.607,171.655,24.909,154.643
C09763=1063.798,-99.985,-60.618,171.657,24.910,154.643
C09764=1063.804,-99.735,-60.627,171.658,24.911,154.643
C09765=1063.810,-99.485,-60.639,171.660,24.912,154.643
C09766=1063.816,-99.235,-60.648,171.662,24.914,154.643
C09767=1063.823,-98.986,-60.658,171.663,24.915,154.643
C09768=1063.829,-98.702,-60.670,171.665,24.916,154.643
C09769=1063.836,-98.418,-60.681,171.668,24.918,154.643
C09770=1063.843,-98.135,-60.693,171.670,24.919,154.643
C09771=1063.850,-97.850,-60.705,171.671,24.920,154.643
C09772=1063.856,-97.600,-60.714,171.673,24.921,154.643
C09773=1063.862,-97.351,-60.725,171.675,24.922,154.643
C09774=1063.869,-97.101,-60.736,171.676,24.924,154.643
C09775=1063.875,-96.851,-60.746,171.678,24.926,154.643
C09776=1063.881,-96.601,-60.756,171.680,24.927,154.643
C09777=1063.887,-96.351,-60.767,171.681,24.928,154.643
C09778=1063.893,-96.102,-60.777,171.683,24.929,154.643
C09779=1063.899,-95.853,-60.788,171.686,24.931,154.643
C09780=1063.904,-95.603,-60.798,171.687,24.932,154.643
C09781=1063.911,-95.353,-60.808,171.689,24.933,154.643
C09782=1063.917,-95.103,-60.819,171.691,24.935,154.643
C09783=1063.923,-94.853,-60.829,171.692,24.936,154.643
C09784=1063.929,-94.604,-60.840,171.694,24.937,154.643
C09785=1063.935,-94.354,-60.849,171.696,24.939,154.643
C09786=1063.941,-94.105,-60.860,171.697,24.940,154.643
C09787=1063.947,-93.854,-60.872,171.699,24.941,154.643
C09788=1063.953,-93.605,-60.881,171.701,24.943,154.643
C09789=1063.959,-93.355,-60.892,171.702,24.944,154.643
C09790=1063.966,-93.106,-60.902,171.704,24.945,154.643
C09791=1063.971,-92.856,-60.912,171.706,24.947,154.643
C09792=1063.977,-92.606,-60.924,171.707,24.948,154.643
C09793=1063.984,-92.356,-60.934,171.709,24.950,154.644
C09794=1063.989,-92.106,-60.944,171.711,24.951,154.644
C09795=1063.996,-91.857,-60.954,171.712,24.952,154.644
C09796=1064.001,-91.608,-60.965,171.714,24.953,154.644
C09797=1064.008,-91.357,-60.977,171.716,24.955,154.644
C09798=1064.014,-91.108,-60.986,171.717,24.956,154.644
C09799=1064.020,-90.858,-60.997,171.719,24.958,154.644
C09800=1064.026,-90.609,-61.007,171.721,24.959,154.644
C09801=1064.033,-90.359,-61.019,171.722,24.961,154.644
C09802=1064.038,-90.109,-61.029,171.724,24.962,154.644
C09803=1064.044,-89.860,-61.039,171.726,24.963,154.644
C09804=1064.050,-89.610,-61.050,171.728,24.965,154.644
C09805=1064.057,-89.360,-61.061,171.730,24.967,154.644
C09806=1064.063,-89.111,-61.071,171.732,24.968,154.644
C09807=1064.068,-88.861,-61.082,171.733,24.969,154.644
C09808=1064.075,-88.611,-61.092,171.735,24.970,154.644
C09809=1064.081,-88.361,-61.103,171.737,24.972,154.644
C09810=1064.087,-88.112,-61.114,171.738,24.973,154.644
C09811=1064.093,-87.863,-61.124,171.740,24.974,154.644
C09812=1064.099,-87.612,-61.135,171.742,24.976,154.644
C09813=1064.105,-87.362,-61.146,171.743,24.978,154.644
C09814=1064.112,-87.113,-61.156,171.745,24.979,154.644
C09815=1064.118,-86.863,-61.167,171.747,24.981,154.645
C09816=1064.124,-86.613,-61.178,171.748,24.982,154.645
C09817=1064.130,-86.364,-61.188,171.750,24.983,154.645
C09818=1064.137,-86.114,-61.200,171.752,24.985,154.645
C09819=1064.142,-85.865,-61.210,171.753,24.986,154.645
C09820=1064.149,-85.615,-61.221,171.755,24.987,154.645
C09821=1064.155,-85.365,-61.231,171.756,24.989,154.645
C09822=1064.161,-85.115,-61.242,171.758,24.990,154.645
C09823=1064.167,-84.866,-61.252,171.760,24.992,154.645
C09824=1064.173,-84.616,-61.264,171.761,24.993,154.645
C09825=1064.179,-84.366,-61.275,171.763,24.995,154.645
C09826=1064.186,-84.116,-61.285,171.766,24.997,154.645
C09827=1064.192,-83.867,-61.296,171.767,24.998,154.645
C09828=1064.198,-83.617,-61.307,171.769,24.999,154.645
C09829=1064.204,-83.367,-61.318,171.771,25.001,154.645
C09830=1064.211,-83.118,-61.328,171.772,25.002,154.645
C09831=1064.216,-82.868,-61.339,171.774,25.004,154.646
C09832=1064.224,-82.586,-61.352,171.776,25.005,154.646
C09833=1064.231,-82.304,-61.364,171.777,25.007,154.646
C09834=1064.238,-82.023,-61.377,171.780,25.009,154.646
C09835=1064.245,-81.742,-61.389,171.781,25.010,154.646
C09836=1064.250,-81.492,-61.399,171.783,25.012,154.646
C09837=1064.258,-81.242,-61.410,171.785,25.013,154.646
C09838=1064.263,-80.993,-61.421,171.786,25.015,154.646
C09839=1064.269,-80.743,-61.432,171.788,25.016,154.646
C09840=1064.275,-80.493,-61.443,171.790,25.018,154.646
C09841=1064.282,-80.244,-61.453,171.791,25.019,154.646
C09842=1064.288,-79.994,-61.465,171.793,25.021,154.646
C09843=1064.294,-79.744,-61.475,171.794,25.023,154.646
C09844=1064.300,-79.494,-61.487,171.796,25.024,154.646
C09845=1064.306,-79.245,-61.498,171.799,25.026,154.647
C09846=1064.312,-78.996,-61.509,171.800,25.028,154.647
C09847=1064.318,-78.746,-61.520,171.802,25.029,154.647
C09848=1064.325,-78.496,-61.531,171.803,25.031,154.647
C09849=1064.331,-78.246,-61.542,171.805,25.032,154.647
C09850=1064.337,-77.997,-61.553,171.807,25.034,154.647
C09851=1064.343,-77.747,-61.564,171.808,25.036,154.647
C09852=1064.349,-77.497,-61.575,171.810,25.037,154.647
C09853=1064.355,-77.248,-61.587,171.812,25.039,154.647
C09854=1064.361,-76.998,-61.598,171.813,25.040,154.647
C09855=1064.367,-76.749,-61.609,171.815,25.042,154.647
C09856=1064.373,-76.498,-61.620,171.816,25.043,154.648
C09857=1064.379,-76.249,-61.631,171.818,25.045,154.648
C09858=1064.386,-75.999,-61.642,171.820,25.046,154.648
C09859=1064.392,-75.750,-61.654,171.821,25.048,154.648
C09860=1064.398,-75.500,-61.665,171.823,25.049,154.648
C09861=1064.404,-75.250,-61.676,171.824,25.051,154.648
C09862=1064.409,-75.001,-61.687,171.826,25.053,154.648
C09863=1064.416,-74.751,-61.699,171.828,25.055,154.648
C09864=1064.422,-74.502,-61.709,171.829,25.056,154.648
C09865=1064.428,-74.251,-61.721,171.831,25.058,154.649
C09866=1064.434,-74.002,-61.732,171.833,25.060,154.649
C09867=1064.441,-73.752,-61.744,171.835,25.061,154.649
C09868=1064.446,-73.503,-61.754,171.837,25.063,154.649
C09869=1064.453,-73.253,-61.766,171.838,25.065,154.649
C09870=1064.458,-73.003,-61.777,171.840,25.067,154.649
C09871=1064.465,-72.754,-61.789,171.841,25.068,154.649
C09872=1064.470,-72.504,-61.800,171.843,25.070,154.649
C09873=1064.476,-72.254,-61.811,171.845,25.071,154.649
C09874=1064.482,-72.005,-61.823,171.846,25.073,154.650
C09875=1064.488,-71.755,-61.834,171.848,25.075,154.650
C09876=1064.494,-71.505,-61.845,171.849,25.077,154.650
C09877=1064.500,-71.256,-61.857,171.851,25.079,154.650
C09878=1064.506,-71.006,-61.868,171.852,25.080,154.650
C09879=1064.512,-70.756,-61.879,171.854,25.082,154.650
C09880=1064.518,-70.507,-61.891,171.856,25.084,154.650
C09881=1064.524,-70.257,-61.902,171.857,25.086,154.650
C09882=1064.530,-70.007,-61.915,171.859,25.087,154.651
C09883=1064.536,-69.758,-61.926,171.860,25.089,154.651
C09884=1064.542,-69.508,-61.937,171.862,25.091,154.651
C09885=1064.548,-69.259,-61.948,171.864,25.092,154.651
C09886=1064.555,-69.008,-61.960,171.865,25.094,154.651
C09887=1064.560,-68.759,-61.972,171.867,25.096,154.651
C09888=1064.566,-68.509,-61.983,171.869,25.098,154.651
C09889=1064.572,-68.260,-61.994,171.871,25.100,154.651
C09890=1064.579,-68.010,-62.006,171.872,25.102,154.652
C09891=1064.584,-67.760,-62.017,171.874,25.104,154.652
C09892=1064.590,-67.511,-62.029,171.875,25.105,154.652
C09893=1064.596,-67.261,-62.040,171.877,25.107,154.652
C09894=1064.603,-67.012,-62.052,171.879,25.109,154.652
C09895=1064.609,-66.761,-62.063,171.880,25.111,154.652
C09896=1064.615,-66.482,-62.076,171.882,25.113,154.652
C09897=1064.622,-66.203,-62.089,171.883,25.114,154.653
C09898=1064.629,-65.923,-62.102,171.886,25.117,154.653
C09899=1064.635,-65.644,-62.115,171.887,25.118,154.653
C09900=1064.642,-65.395,-62.127,171.889,25.120,154.653
C09901=1064.647,-65.145,-62.138,171.890,25.122,154.653
C09902=1064.654,-64.895,-62.150,171.892,25.124,154.653
C09903=1064.660,-64.646,-62.162,171.894,25.126,154.653
C09904=1064.666,-64.396,-62.173,171.895,25.127,154.654
C09905=1064.672,-64.146,-62.186,171.897,25.129,154.654
C09906=1064.678,-63.897,-62.197,171.898,25.131,154.654
C09907=1064.684,-63.647,-62.209,171.900,25.133,154.654
C09908=1064.690,-63.397,-62.221,171.901,25.134,154.654
C09909=1064.696,-63.148,-62.232,171.903,25.136,154.654
C09910=1064.703,-62.898,-62.244,171.906,25.138,154.654
C09911=1064.709,-62.648,-62.255,171.907,25.140,154.654
C09912=1064.714,-62.399,-62.267,171.909,25.142,154.655
C09913=1064.721,-62.149,-62.279,171.910,25.144,154.655
C09914=1064.727,-61.900,-62.290,171.912,25.146,154.655
C09915=1064.733,-61.650,-62.303,171.913,25.148,154.655
C09916=1064.739,-61.400,-62.314,171.915,25.150,154.655
C09917=1064.745,-61.151,-62.326,171.916,25.152,154.655
C09918=1064.751,-60.901,-62.338,171.918,25.153,154.656
C09919=1064.757,-60.651,-62.350,171.920,25.155,154.656
C09920=1064.763,-60.402,-62.361,171.921,25.157,154.656
C09921=1064.770,-60.152,-62.373,171.923,25.159,154.656
C09922=1064.776,-59.902,-62.385,171.924,25.161,154.656
C09923=1064.782,-59.652,-62.397,171.926,25.162,154.656
C09924=1064.788,-59.403,-62.408,171.927,25.164,154.656
C09925=1064.794,-59.153,-62.420,171.929,25.166,154.657
C09926=1064.800,-58.903,-62.432,171.930,25.168,154.657
C09927=1064.807,-58.654,-62.444,171.932,25.170,154.657
C09928=1064.812,-58.405,-62.456,171.934,25.171,154.657
C09929=1064.819,-58.154,-62.468,171.935,25.174,154.657
C09930=1064.825,-57.905,-62.479,171.937,25.175,154.657
C09931=1064.831,-57.656,-62.492,171.938,25.177,154.658
C09932=1064.837,-57.406,-62.504,171.941,25.179,154.658
C09933=1064.844,-57.156,-62.515,171.942,25.181,154.658
C09934=1064.849,-56.907,-62.527,171.944,25.183,154.658
C09935=1064.856,-56.657,-62.539,171.945,25.185,154.658
C09936=1064.862,-56.408,-62.551,171.947,25.187,154.658
C09937=1064.868,-56.158,-62.564,171.948,25.189,154.659
C09938=1064.874,-55.908,-62.575,171.950,25.191,154.659
C09939=1064.880,-55.658,-62.587,171.952,25.193,154.659
C09940=1064.887,-55.409,-62.599,171.953,25.194,154.659
C09941=1064.893,-55.159,-62.611,171.955,25.196,154.659
C09942=1064.899,-54.909,-62.624,171.956,25.198,154.659
C09943=1064.905,-54.660,-62.634,171.958,25.200,154.659
C09944=1064.911,-54.410,-62.646,171.959,25.202,154.660
C09945=1064.917,-54.160,-62.659,171.961,25.204,154.660
C09946=1064.924,-53.911,-62.671,171.962,25.206,154.660
C09947=1064.930,-53.661,-62.683,171.964,25.207,154.660
C09948=1064.936,-53.412,-62.695,171.966,25.209,154.660
C09949=1064.943,-53.162,-62.707,171.967,25.211,154.660
C09950=1064.949,-52.913,-62.720,171.969,25.213,154.661
C09951=1064.955,-52.663,-62.732,171.970,25.215,154.661
C09952=1064.962,-52.413,-62.743,171.972,25.217,154.661
C09953=1064.967,-52.164,-62.755,171.973,25.219,154.661
C09954=1064.973,-51.914,-62.767,171.976,25.221,154.661
C09955=1064.979,-51.664,-62.779,171.977,25.223,154.661
C09956=1064.986,-51.415,-62.791,171.979,25.225,154.662
C09957=1064.992,-51.165,-62.804,171.980,25.227,154.662
C09958=1064.999,-50.915,-62.816,171.982,25.229,154.662
C09959=1065.005,-50.665,-62.828,171.984,25.230,154.662
C09960=1065.012,-50.387,-62.841,171.985,25.233,154.662
C09961=1065.019,-50.109,-62.856,171.987,25.235,154.662
C09962=1065.025,-49.832,-62.869,171.989,25.237,154.663
C09963=1065.031,-49.553,-62.882,171.990,25.240,154.663
C09964=1065.037,-49.304,-62.895,171.992,25.241,154.663
C09965=1065.044,-49.054,-62.907,171.993,25.244,154.663
C09966=1065.050,-48.805,-62.920,171.995,25.246,154.663
C09967=1065.056,-48.555,-62.932,171.997,25.247,154.664
C09968=1065.062,-48.306,-62.944,171.998,25.250,154.664
C09969=1065.068,-48.056,-62.957,172.000,25.252,154.664
C09970=1065.074,-47.806,-62.969,172.001,25.254,154.664
C09971=1065.080,-47.556,-62.982,172.003,25.256,154.664
C09972=1065.086,-47.307,-62.994,172.004,25.258,154.665
C09973=1065.092,-47.057,-63.006,172.006,25.260,154.665
C09974=1065.098,-46.808,-63.018,172.007,25.262,154.665
C09975=1065.104,-46.558,-63.030,172.009,25.264,154.665
C09976=1065.110,-46.308,-63.043,172.010,25.266,154.665
C09977=1065.116,-46.058,-63.055,172.012,25.268,154.666
C09978=1065.122,-45.809,-63.069,172.013,25.270,154.666
C09979=1065.129,-45.560,-63.081,172.015,25.272,154.666
C09980=1065.134,-45.310,-63.093,172.016,25.274,154.666
C09981=1065.140,-45.060,-63.105,172.019,25.277,154.666
C09982=1065.146,-44.811,-63.118,172.020,25.279,154.667
C09983=1065.153,-44.561,-63.130,172.022,25.281,154.667
C09984=1065.159,-44.311,-63.142,172.023,25.283,154.667
C09985=1065.165,-44.062,-63.156,172.025,25.284,154.667
C09986=1065.172,-43.812,-63.168,172.026,25.287,154.667
C09987=1065.177,-43.562,-63.180,172.028,25.289,154.668
C09988=1065.183,-43.313,-63.193,172.029,25.291,154.668
C09989=1065.189,-43.063,-63.205,172.031,25.293,154.668
C09990=1065.196,-42.814,-63.218,172.032,25.295,154.668
C09991=1065.202,-42.565,-63.230,172.034,25.297,154.668
C09992=1065.207,-42.315,-63.243,172.035,25.299,154.669
C09993=1065.213,-42.065,-63.255,172.037,25.301,154.669
C09994=1065.220,-41.815,-63.269,172.038,25.303,154.669
C09995=1065.226,-41.566,-63.281,172.040,25.305,154.669
C09996=1065.232,-41.316,-63.293,172.041,25.308,154.669
//INST
///DATE 2021/06/17 10:55
///ATTR SC,RW,RJ
////FRAME ROBOT
///GROUP1 RB1
NOP
MOVL C00000 V=800.0 PL=0
MOVL C00001 V=800.0 PL=0
MOVL C00002 V=800.0 PL=0
MOVL C00003 V=800.0 PL=0
MOVL C00004 V=800.0 PL=0
MOVL C00005 V=800.0 PL=0
MOVL C00006 V=800.0 PL=0
MOVL C00007 V=800.0 PL=0
MOVL C00008 V=800.0 PL=0
MOVL C00009 V=800.0 PL=0
MOVL C00010 V=800.0 PL=0
MOVL C00011 V=800.0 PL=0
MOVL C00012 V=800.0 PL=0
MOVL C00013 V=800.0 PL=0
MOVL C00014 V=800.0 PL=0
MOVL C00015 V=800.0 PL=0
MOVL C00016 V=800.0 PL=0
MOVL C00017 V=800.0 PL=0
MOVL C00018 V=800.0 PL=0
MOVL C00019 V=800.0 PL=0
MOVL C00020 V=800.0 PL=0
MOVL C00021 V=800.0 PL=0
MOVL C00022 V=800.0 PL=0
MOVL C00023 V=800.0 PL=0
MOVL C00024 V=800.0 PL=0
MOVL C00025 V=800.0 PL=0
MOVL C00026 V=800.0 PL=0
MOVL C00027 V=800.0 PL=0
MOVL C00028 V=800.0 PL=0
MOVL C00029 V=800.0 PL=0
MOVL C00030 V=800.0 PL=0
MOVL C00031 V=800.0 PL=0
MOVL C00032 V=800.0 PL=0
MOVL C00033 V=800.0 PL=0
MOVL C00034 V=800.0 PL=0
MOVL C00035 V=800.0 PL=0
MOVL C00036 V=800.0 PL=0
MOVL C00037 V=800.0 PL=0
MOVL C00038 V=800.0 PL=0
MOVL C00039 V=800.0 PL=0
MOVL C00040 V=800.0 PL=0
MOVL C00041 V=800.0 PL=0
MOVL C00042 V=800.0 PL=0
MOVL C00043 V=800.0 PL=0
MOVL C00044 V=800.0 PL=0
MOVL C00045 V=800.0 PL=0
MOVL C00046 V=800.0 PL=0
MOVL C00047 V=800.0 PL=0
MOVL C00048 V=800.0 PL=0
MOVL C00049 V=800.0 PL=0
MOVL C00050 V=800.0 PL=0
MOVL C00051 V=800.0 PL=0
MOVL C00052 V=800.0 PL=0
MOVL C00053 V=800.0 PL=0
MOVL C00054 V=800.0 PL=0
MOVL C00055 V=800.0 PL=0
MOVL C00056 V=800.0 PL=0
MOVL C00057 V=800.0 PL=0
MOVL C00058 V=800.0 PL=0
MOVL C00059 V=800.0 PL=0
MOVL C00060 V=800.0 PL=0
MOVL C00061 V=800.0 PL=0
MOVL C00062 V=800.0 PL=0
MOVL C00063 V=800.0 PL=0
MOVL C00064 V=800.0 PL=0
MOVL C00065 V=800.0 PL=0
MOVL C00066 V=800.0 PL=0
MOVL C00067 V=800.0 PL=0
MOVL C00068 V=800.0 PL=0
MOVL C00069 V=800.0 PL=0
MOVL C00070 V=800.0 PL=0
MOVL C00071 V=800.0 PL=0
MOVL C00072 V=800.0 PL=0
MOVL C00073 V=800.0 PL=0
MOVL C00074 V=800.0 PL=0
MOVL C00075 V=800.0 PL=0
MOVL C00076 V=800.0 PL=0
MOVL C00077 V=800.0 PL=0
MOVL C00078 V=800.0 PL=0
MOVL C00079 V=800.0 PL=0
MOVL C00080 V=800.0 PL=0
MOVL C00081 V=800.0 PL=0
MOVL C00082 V=800.0 PL=0
MOVL C00083 V=800.0 PL=0
MOVL C00084 V=800.0 PL=0
MOVL C00085 V=800.0 PL=0
MOVL C00086 V=800.0 PL=0
MOVL C00087 V=800.0 PL=0
MOVL C00088 V=800.0 PL=0
MOVL C00089 V=800.0 PL=0
MOVL C00090 V=800.0 PL=0
MOVL C00091 V=800.0 PL=0
MOVL C00092 V=800.0 PL=0
MOVL C00093 V=800.0 PL=0
MOVL C00094 V=800.0 PL=0
MOVL C00095 V=800.0 PL=0
MOVL C00096 V=800.0 PL=0
MOVL C00097 V=800.0 PL=0
MOVL C00098 V=800.0 PL=0
MOVL C00099 V=800.0 PL=0
MOVL C00100 V=800.0 PL=0
MOVL C00101 V=800.0 PL=0
MOVL C00102 V=800.0 PL=0
MOVL C00103 V=800.0 PL=0
MOVL C00104 V=800.0 PL=0
MOVL C00105 V=800.0 PL=0
MOVL C00106 V=800.0 PL=0
MOVL C00107 V=800.0 PL=0
MOVL C00108 V=800.0 PL=0
MOVL C00109 V=800.0 PL=0
MOVL C00110 V=800.0 PL=0
MOVL C00111 V=800.0 PL=0
MOVL C00112 V=800.0 PL=0
MOVL C00113 V=800.0 PL=0
MOVL C00114 V=800.0 PL=0
MOVL C00115 V=800.0 PL=0
MOVL C00116 V=800.0 PL=0
MOVL C00117 V=800.0 PL=0
MOVL C00118 V=800.0 PL=0
MOVL C00119 V=800.0 PL=0
MOVL C00120 V=800.0 PL=0
MOVL C00121 V=800.0 PL=0
MOVL C00122 V=800.0 PL=0
MOVL C00123 V=800.0 PL=0
MOVL C00124 V=800.0 PL=0
MOVL C00125 V=800.0 PL=0
MOVL C00126 V=800.0 PL=0
MOVL C00127 V=800.0 PL=0
MOVL C00128 V=800.0 PL=0
MOVL C00129 V=800.0 PL=0
MOVL C00130 V=800.0 PL=0
MOVL C00131 V=800.0 PL=0
MOVL C00132 V=800.0 PL=0
MOVL C00133 V=800.0 PL=0
MOVL C00134 V=800.0 PL=0
MOVL C00135 V=800.0 PL=0
MOVL C00136 V=800.0 PL=0
MOVL C00137 V=800.0 PL=0
MOVL C00138 V=800.0 PL=0
MOVL C00139 V=800.0 PL=0
MOVL C00140 V=800.0 PL=0
MOVL C00141 V=800.0 PL=0
MOVL C00142 V=800.0 PL=0
MOVL C00143 V=800.0 PL=0
MOVL C00144 V=800.0 PL=0
MOVL C00145 V=800.0 PL=0
MOVL C00146 V=800.0 PL=0
MOVL C00147 V=800.0 PL=0
MOVL C00148 V=800.0 PL=0
MOVL C00149 V=800.0 PL=0
MOVL C00150 V=800.0 PL=0
MOVL C00151 V=800.0 PL=0
MOVL C00152 V=800.0 PL=0
MOVL C00153 V=800.0 PL=0
MOVL C00154 V=800.0 PL=0
MOVL C00155 V=800.0 PL=0
MOVL C00156 V=800.0 PL=0
MOVL C00157 V=800.0 PL=0
MOVL C00158 V=800.0 PL=0
MOVL C00159 V=800.0 PL=0
MOVL C00160 V=800.0 PL=0
MOVL C00161 V=800.0 PL=0
MOVL C00162 V=800.0 PL=0
MOVL C00163 V=800.0 PL=0
MOVL C00164 V=800.0 PL=0
MOVL C00165 V=800.0 PL=0
MOVL C00166 V=800.0 PL=0
MOVL C00167 V=800.0 PL=0
MOVL C00168 V=800.0 PL=0
MOVL C00169 V=800.0 PL=0
MOVL C00170 V=800.0 PL=0
MOVL C00171 V=800.0 PL=0
MOVL C00172 V=800.0 PL=0
MOVL C00173 V=800.0 PL=0
MOVL C00174 V=800.0 PL=0
MOVL C00175 V=800.0 PL=0
MOVL C00176 V=800.0 PL=0
MOVL C00177 V=800.0 PL=0
MOVL C00178 V=800.0 PL=0
MOVL C00179 V=800.0 PL=0
MOVL C00180 V=800.0 PL=0
MOVL C00181 V=800.0 PL=0
MOVL C00182 V=800.0 PL=0
MOVL C00183 V=800.0 PL=0
MOVL C00184 V=800.0 PL=0
MOVL C00185 V=800.0 PL=0
MOVL C00186 V=800.0 PL=0
MOVL C00187 V=800.0 PL=0
MOVL C00188 V=800.0 PL=0
MOVL C00189 V=800.0 PL=0
MOVL C00190 V=800.0 PL=0
MOVL C00191 V=800.0 PL=0
MOVL C00192 V=800.0 PL=0
MOVL C00193 V=800.0 PL=0
MOVL C00194 V=800.0 PL=0
MOVL C00195 V=800.0 PL=0
MOVL C00196 V=800.0 PL=0
MOVL C00197 V=800.0 PL=0
MOVL C00198 V=800.0 PL=0
MOVL C00199 V=800.0 PL=0
MOVL C00200 V=800.0 PL=0
MOVL C00201 V=800.0 PL=0
MOVL C00202 V=800.0 PL=0
MOVL C00203 V=800.0 PL=0
MOVL C00204 V=800.0 PL=0
MOVL C00205 V=800.0 PL=0
MOVL C00206 V=800.0 PL=0
MOVL C00207 V=800.0 PL=0
MOVL C00208 V=800.0 PL=0
MOVL C00209 V=800.0 PL=0
MOVL C00210 V=800.0 PL=0
MOVL C00211 V=800.0 PL=0
MOVL C00212 V=800.0 PL=0
MOVL C00213 V=800.0 PL=0
MOVL C00214 V=800.0 PL=0
MOVL C00215 V=800.0 PL=0
MOVL C00216 V=800.0 PL=0
MOVL C00217 V=800.0 PL=0
MOVL C00218 V=800.0 PL=0
MOVL C00219 V=800.0 PL=0
MOVL C00220 V=800.0 PL=0
MOVL C00221 V=800.0 PL=0
MOVL C00222 V=800.0 PL=0
MOVL C00223 V=800.0 PL=0
MOVL C00224 V=800.0 PL=0
MOVL C00225 V=800.0 PL=0
MOVL C00226 V=800.0 PL=0
MOVL C00227 V=800.0 PL=0
MOVL C00228 V=800.0 PL=0
MOVL C00229 V=800.0 PL=0
MOVL C00230 V=800.0 PL=0
MOVL C00231 V=800.0 PL=0
MOVL C00232 V=800.0 PL=0
MOVL C00233 V=800.0 PL=0
MOVL C00234 V=800.0 PL=0
MOVL C00235 V=800.0 PL=0
MOVL C00236 V=800.0 PL=0
MOVL C00237 V=800.0 PL=0
MOVL C00238 V=800.0 PL=0
MOVL C00239 V=800.0 PL=0
MOVL C00240 V=800.0 PL=0
MOVL C00241 V=800.0 PL=0
MOVL C00242 V=800.0 PL=0
MOVL C00243 V=800.0 PL=0
MOVL C00244 V=800.0 PL=0
MOVL C00245 V=800.0 PL=0
MOVL C00246 V=800.0 PL=0
MOVL C00247 V=800.0 PL=0
MOVL C00248 V=800.0 PL=0
MOVL C00249 V=800.0 PL=0
MOVL C00250 V=800.0 PL=0
MOVL C00251 V=800.0 PL=0
MOVL C00252 V=800.0 PL=0
MOVL C00253 V=800.0 PL=0
MOVL C00254 V=800.0 PL=0
MOVL C00255 V=800.0 PL=0
MOVL C00256 V=800.0 PL=0
MOVL C00257 V=800.0 PL=0
MOVL C00258 V=800.0 PL=0
MOVL C00259 V=800.0 PL=0
MOVL C00260 V=800.0 PL=0
MOVL C00261 V=800.0 PL=0
MOVL C00262 V=800.0 PL=0
MOVL C00263 V=800.0 PL=0
MOVL C00264 V=800.0 PL=0
MOVL C00265 V=800.0 PL=0
MOVL C00266 V=800.0 PL=0
MOVL C00267 V=800.0 PL=0
MOVL C00268 V=800.0 PL=0
MOVL C00269 V=800.0 PL=0
MOVL C00270 V=800.0 PL=0
MOVL C00271 V=800.0 PL=0
MOVL C00272 V=800.0 PL=0
MOVL C00273 V=800.0 PL=0
MOVL C00274 V=800.0 PL=0
MOVL C00275 V=800.0 PL=0
MOVL C00276 V=800.0 PL=0
MOVL C00277 V=800.0 PL=0
MOVL C00278 V=800.0 PL=0
MOVL C00279 V=800.0 PL=0
MOVL C00280 V=800.0 PL=0
MOVL C00281 V=800.0 PL=0
MOVL C00282 V=800.0 PL=0
MOVL C00283 V=800.0 PL=0
MOVL C00284 V=800.0 PL=0
MOVL C00285 V=800.0 PL=0
MOVL C00286 V=800.0 PL=0
MOVL C00287 V=800.0 PL=0
MOVL C00288 V=800.0 PL=0
MOVL C00289 V=800.0 PL=0
MOVL C00290 V=800.0 PL=0
MOVL C00291 V=800.0 PL=0
MOVL C00292 V=800.0 PL=0
MOVL C00293 V=800.0 PL=0
MOVL C00294 V=800.0 PL=0
MOVL C00295 V=800.0 PL=0
MOVL C00296 V=800.0 PL=0
MOVL C00297 V=800.0 PL=0
MOVL C00298 V=800.0 PL=0
MOVL C00299 V=800.0 PL=0
MOVL C00300 V=800.0 PL=0
MOVL C00301 V=800.0 PL=0
MOVL C00302 V=800.0 PL=0
MOVL C00303 V=800.0 PL=0
MOVL C00304 V=800.0 PL=0
MOVL C00305 V=800.0 PL=0
MOVL C00306 V=800.0 PL=0
MOVL C00307 V=800.0 PL=0
MOVL C00308 V=800.0 PL=0
MOVL C00309 V=800.0 PL=0
MOVL C00310 V=800.0 PL=0
MOVL C00311 V=800.0 PL=0
MOVL C00312 V=800.0 PL=0
MOVL C00313 V=800.0 PL=0
MOVL C00314 V=800.0 PL=0
MOVL C00315 V=800.0 PL=0
MOVL C00316 V=800.0 PL=0
MOVL C00317 V=800.0 PL=0
MOVL C00318 V=800.0 PL=0
MOVL C00319 V=800.0 PL=0
MOVL C00320 V=800.0 PL=0
MOVL C00321 V=800.0 PL=0
MOVL C00322 V=800.0 PL=0
MOVL C00323 V=800.0 PL=0
MOVL C00324 V=800.0 PL=0
MOVL C00325 V=800.0 PL=0
MOVL C00326 V=800.0 PL=0
MOVL C00327 V=800.0 PL=0
MOVL C00328 V=800.0 PL=0
MOVL C00329 V=800.0 PL=0
MOVL C00330 V=800.0 PL=0
MOVL C00331 V=800.0 PL=0
MOVL C00332 V=800.0 PL=0
MOVL C00333 V=800.0 PL=0
MOVL C00334 V=800.0 PL=0
MOVL C00335 V=800.0 PL=0
MOVL C00336 V=800.0 PL=0
MOVL C00337 V=800.0 PL=0
MOVL C00338 V=800.0 PL=0
MOVL C00339 V=800.0 PL=0
MOVL C00340 V=800.0 PL=0
MOVL C00341 V=800.0 PL=0
MOVL C00342 V=800.0 PL=0
MOVL C00343 V=800.0 PL=0
MOVL C00344 V=800.0 PL=0
MOVL C00345 V=800.0 PL=0
MOVL C00346 V=800.0 PL=0
MOVL C00347 V=800.0 PL=0
MOVL C00348 V=800.0 PL=0
MOVL C00349 V=800.0 PL=0
MOVL C00350 V=800.0 PL=0
MOVL C00351 V=800.0 PL=0
MOVL C00352 V=800.0 PL=0
MOVL C00353 V=800.0 PL=0
MOVL C00354 V=800.0 PL=0
MOVL C00355 V=800.0 PL=0
MOVL C00356 V=800.0 PL=0
MOVL C00357 V=800.0 PL=0
MOVL C00358 V=800.0 PL=0
MOVL C00359 V=800.0 PL=0
MOVL C00360 V=800.0 PL=0
MOVL C00361 V=800.0 PL=0
MOVL C00362 V=800.0 PL=0
MOVL C00363 V=800.0 PL=0
MOVL C00364 V=800.0 PL=0
MOVL C00365 V=800.0 PL=0
MOVL C00366 V=800.0 PL=0
MOVL C00367 V=800.0 PL=0
MOVL C00368 V=800.0 PL=0
MOVL C00369 V=800.0 PL=0
MOVL C00370 V=800.0 PL=0
MOVL C00371 V=800.0 PL=0
MOVL C00372 V=800.0 PL=0
MOVL C00373 V=800.0 PL=0
MOVL C00374 V=800.0 PL=0
MOVL C00375 V=800.0 PL=0
MOVL C00376 V=800.0 PL=0
MOVL C00377 V=800.0 PL=0
MOVL C00378 V=800.0 PL=0
MOVL C00379 V=800.0 PL=0
MOVL C00380 V=800.0 PL=0
MOVL C00381 V=800.0 PL=0
MOVL C00382 V=800.0 PL=0
MOVL C00383 V=800.0 PL=0
MOVL C00384 V=800.0 PL=0
MOVL C00385 V=800.0 PL=0
MOVL C00386 V=800.0 PL=0
MOVL C00387 V=800.0 PL=0
MOVL C00388 V=800.0 PL=0
MOVL C00389 V=800.0 PL=0
MOVL C00390 V=800.0 PL=0
MOVL C00391 V=800.0 PL=0
MOVL C00392 V=800.0 PL=0
MOVL C00393 V=800.0 PL=0
MOVL C00394 V=800.0 PL=0
MOVL C00395 V=800.0 PL=0
MOVL C00396 V=800.0 PL=0
MOVL C00397 V=800.0 PL=0
MOVL C00398 V=800.0 PL=0
MOVL C00399 V=800.0 PL=0
MOVL C00400 V=800.0 PL=0
MOVL C00401 V=800.0 PL=0
MOVL C00402 V=800.0 PL=0
MOVL C00403 V=800.0 PL=0
MOVL C00404 V=800.0 PL=0
MOVL C00405 V=800.0 PL=0
MOVL C00406 V=800.0 PL=0
MOVL C00407 V=800.0 PL=0
MOVL C00408 V=800.0 PL=0
MOVL C00409 V=800.0 PL=0
MOVL C00410 V=800.0 PL=0
MOVL C00411 V=800.0 PL=0
MOVL C00412 V=800.0 PL=0
MOVL C00413 V=800.0 PL=0
MOVL C00414 V=800.0 PL=0
MOVL C00415 V=800.0 PL=0
MOVL C00416 V=800.0 PL=0
MOVL C00417 V=800.0 PL=0
MOVL C00418 V=800.0 PL=0
MOVL C00419 V=800.0 PL=0
MOVL C00420 V=800.0 PL=0
MOVL C00421 V=800.0 PL=0
MOVL C00422 V=800.0 PL=0
MOVL C00423 V=800.0 PL=0
MOVL C00424 V=800.0 PL=0
MOVL C00425 V=800.0 PL=0
MOVL C00426 V=800.0 PL=0
MOVL C00427 V=800.0 PL=0
MOVL C00428 V=800.0 PL=0
MOVL C00429 V=800.0 PL=0
MOVL C00430 V=800.0 PL=0
MOVL C00431 V=800.0 PL=0
MOVL C00432 V=800.0 PL=0
MOVL C00433 V=800.0 PL=0
MOVL C00434 V=800.0 PL=0
MOVL C00435 V=800.0 PL=0
MOVL C00436 V=800.0 PL=0
MOVL C00437 V=800.0 PL=0
MOVL C00438 V=800.0 PL=0
MOVL C00439 V=800.0 PL=0
MOVL C00440 V=800.0 PL=0
MOVL C00441 V=800.0 PL=0
MOVL C00442 V=800.0 PL=0
MOVL C00443 V=800.0 PL=0
MOVL C00444 V=800.0 PL=0
MOVL C00445 V=800.0 PL=0
MOVL C00446 V=800.0 PL=0
MOVL C00447 V=800.0 PL=0
MOVL C00448 V=800.0 PL=0
MOVL C00449 V=800.0 PL=0
MOVL C00450 V=800.0 PL=0
MOVL C00451 V=800.0 PL=0
MOVL C00452 V=800.0 PL=0
MOVL C00453 V=800.0 PL=0
MOVL C00454 V=800.0 PL=0
MOVL C00455 V=800.0 PL=0
MOVL C00456 V=800.0 PL=0
MOVL C00457 V=800.0 PL=0
MOVL C00458 V=800.0 PL=0
MOVL C00459 V=800.0 PL=0
MOVL C00460 V=800.0 PL=0
MOVL C00461 V=800.0 PL=0
MOVL C00462 V=800.0 PL=0
MOVL C00463 V=800.0 PL=0
MOVL C00464 V=800.0 PL=0
MOVL C00465 V=800.0 PL=0
MOVL C00466 V=800.0 PL=0
MOVL C00467 V=800.0 PL=0
MOVL C00468 V=800.0 PL=0
MOVL C00469 V=800.0 PL=0
MOVL C00470 V=800.0 PL=0
MOVL C00471 V=800.0 PL=0
MOVL C00472 V=800.0 PL=0
MOVL C00473 V=800.0 PL=0
MOVL C00474 V=800.0 PL=0
MOVL C00475 V=800.0 PL=0
MOVL C00476 V=800.0 PL=0
MOVL C00477 V=800.0 PL=0
MOVL C00478 V=800.0 PL=0
MOVL C00479 V=800.0 PL=0
MOVL C00480 V=800.0 PL=0
MOVL C00481 V=800.0 PL=0
MOVL C00482 V=800.0 PL=0
MOVL C00483 V=800.0 PL=0
MOVL C00484 V=800.0 PL=0
MOVL C00485 V=800.0 PL=0
MOVL C00486 V=800.0 PL=0
MOVL C00487 V=800.0 PL=0
MOVL C00488 V=800.0 PL=0
MOVL C00489 V=800.0 PL=0
MOVL C00490 V=800.0 PL=0
MOVL C00491 V=800.0 PL=0
MOVL C00492 V=800.0 PL=0
MOVL C00493 V=800.0 PL=0
MOVL C00494 V=800.0 PL=0
MOVL C00495 V=800.0 PL=0
MOVL C00496 V=800.0 PL=0
MOVL C00497 V=800.0 PL=0
MOVL C00498 V=800.0 PL=0
MOVL C00499 V=800.0 PL=0
MOVL C00500 V=800.0 PL=0
MOVL C00501 V=800.0 PL=0
MOVL C00502 V=800.0 PL=0
MOVL C00503 V=800.0 PL=0
MOVL C00504 V=800.0 PL=0
MOVL C00505 V=800.0 PL=0
MOVL C00506 V=800.0 PL=0
MOVL C00507 V=800.0 PL=0
MOVL C00508 V=800.0 PL=0
MOVL C00509 V=800.0 PL=0
MOVL C00510 V=800.0 PL=0
MOVL C00511 V=800.0 PL=0
MOVL C00512 V=800.0 PL=0
MOVL C00513 V=800.0 PL=0
MOVL C00514 V=800.0 PL=0
MOVL C00515 V=800.0 PL=0
MOVL C00516 V=800.0 PL=0
MOVL C00517 V=800.0 PL=0
MOVL C00518 V=800.0 PL=0
MOVL C00519 V=800.0 PL=0
MOVL C00520 V=800.0 PL=0
MOVL C00521 V=800.0 PL=0
MOVL C00522 V=800.0 PL=0
MOVL C00523 V=800.0 PL=0
MOVL C00524 V=800.0 PL=0
MOVL C00525 V=800.0 PL=0
MOVL C00526 V=800.0 PL=0
MOVL C00527 V=800.0 PL=0
MOVL C00528 V=800.0 PL=0
MOVL C00529 V=800.0 PL=0
MOVL C00530 V=800.0 PL=0
MOVL C00531 V=800.0 PL=0
MOVL C00532 V=800.0 PL=0
MOVL C00533 V=800.0 PL=0
MOVL C00534 V=800.0 PL=0
MOVL C00535 V=800.0 PL=0
MOVL C00536 V=800.0 PL=0
MOVL C00537 V=800.0 PL=0
MOVL C00538 V=800.0 PL=0
MOVL C00539 V=800.0 PL=0
MOVL C00540 V=800.0 PL=0
MOVL C00541 V=800.0 PL=0
MOVL C00542 V=800.0 PL=0
MOVL C00543 V=800.0 PL=0
MOVL C00544 V=800.0 PL=0
MOVL C00545 V=800.0 PL=0
MOVL C00546 V=800.0 PL=0
MOVL C00547 V=800.0 PL=0
MOVL C00548 V=800.0 PL=0
MOVL C00549 V=800.0 PL=0
MOVL C00550 V=800.0 PL=0
MOVL C00551 V=800.0 PL=0
MOVL C00552 V=800.0 PL=0
MOVL C00553 V=800.0 PL=0
MOVL C00554 V=800.0 PL=0
MOVL C00555 V=800.0 PL=0
MOVL C00556 V=800.0 PL=0
MOVL C00557 V=800.0 PL=0
MOVL C00558 V=800.0 PL=0
MOVL C00559 V=800.0 PL=0
MOVL C00560 V=800.0 PL=0
MOVL C00561 V=800.0 PL=0
MOVL C00562 V=800.0 PL=0
MOVL C00563 V=800.0 PL=0
MOVL C00564 V=800.0 PL=0
MOVL C00565 V=800.0 PL=0
MOVL C00566 V=800.0 PL=0
MOVL C00567 V=800.0 PL=0
MOVL C00568 V=800.0 PL=0
MOVL C00569 V=800.0 PL=0
MOVL C00570 V=800.0 PL=0
MOVL C00571 V=800.0 PL=0
MOVL C00572 V=800.0 PL=0
MOVL C00573 V=800.0 PL=0
MOVL C00574 V=800.0 PL=0
MOVL C00575 V=800.0 PL=0
MOVL C00576 V=800.0 PL=0
MOVL C00577 V=800.0 PL=0
MOVL C00578 V=800.0 PL=0
MOVL C00579 V=800.0 PL=0
MOVL C00580 V=800.0 PL=0
MOVL C00581 V=800.0 PL=0
MOVL C00582 V=800.0 PL=0
MOVL C00583 V=800.0 PL=0
MOVL C00584 V=800.0 PL=0
MOVL C00585 V=800.0 PL=0
MOVL C00586 V=800.0 PL=0
MOVL C00587 V=800.0 PL=0
MOVL C00588 V=800.0 PL=0
MOVL C00589 V=800.0 PL=0
MOVL C00590 V=800.0 PL=0
MOVL C00591 V=800.0 PL=0
MOVL C00592 V=800.0 PL=0
MOVL C00593 V=800.0 PL=0
MOVL C00594 V=800.0 PL=0
MOVL C00595 V=800.0 PL=0
MOVL C00596 V=800.0 PL=0
MOVL C00597 V=800.0 PL=0
MOVL C00598 V=800.0 PL=0
MOVL C00599 V=800.0 PL=0
MOVL C00600 V=800.0 PL=0
MOVL C00601 V=800.0 PL=0
MOVL C00602 V=800.0 PL=0
MOVL C00603 V=800.0 PL=0
MOVL C00604 V=800.0 PL=0
MOVL C00605 V=800.0 PL=0
MOVL C00606 V=800.0 PL=0
MOVL C00607 V=800.0 PL=0
MOVL C00608 V=800.0 PL=0
MOVL C00609 V=800.0 PL=0
MOVL C00610 V=800.0 PL=0
MOVL C00611 V=800.0 PL=0
MOVL C00612 V=800.0 PL=0
MOVL C00613 V=800.0 PL=0
MOVL C00614 V=800.0 PL=0
MOVL C00615 V=800.0 PL=0
MOVL C00616 V=800.0 PL=0
MOVL C00617 V=800.0 PL=0
MOVL C00618 V=800.0 PL=0
MOVL C00619 V=800.0 PL=0
MOVL C00620 V=800.0 PL=0
MOVL C00621 V=800.0 PL=0
MOVL C00622 V=800.0 PL=0
MOVL C00623 V=800.0 PL=0
MOVL C00624 V=800.0 PL=0
MOVL C00625 V=800.0 PL=0
MOVL C00626 V=800.0 PL=0
MOVL C00627 V=800.0 PL=0
MOVL C00628 V=800.0 PL=0
MOVL C00629 V=800.0 PL=0
MOVL C00630 V=800.0 PL=0
MOVL C00631 V=800.0 PL=0
MOVL C00632 V=800.0 PL=0
MOVL C00633 V=800.0 PL=0
MOVL C00634 V=800.0 PL=0
MOVL C00635 V=800.0 PL=0
MOVL C00636 V=800.0 PL=0
MOVL C00637 V=800.0 PL=0
MOVL C00638 V=800.0 PL=0
MOVL C00639 V=800.0 PL=0
MOVL C00640 V=800.0 PL=0
MOVL C00641 V=800.0 PL=0
MOVL C00642 V=800.0 PL=0
MOVL C00643 V=800.0 PL=0
MOVL C00644 V=800.0 PL=0
MOVL C00645 V=800.0 PL=0
MOVL C00646 V=800.0 PL=0
MOVL C00647 V=800.0 PL=0
MOVL C00648 V=800.0 PL=0
MOVL C00649 V=800.0 PL=0
MOVL C00650 V=800.0 PL=0
MOVL C00651 V=800.0 PL=0
MOVL C00652 V=800.0 PL=0
MOVL C00653 V=800.0 PL=0
MOVL C00654 V=800.0 PL=0
MOVL C00655 V=800.0 PL=0
MOVL C00656 V=800.0 PL=0
MOVL C00657 V=800.0 PL=0
MOVL C00658 V=800.0 PL=0
MOVL C00659 V=800.0 PL=0
MOVL C00660 V=800.0 PL=0
MOVL C00661 V=800.0 PL=0
MOVL C00662 V=800.0 PL=0
MOVL C00663 V=800.0 PL=0
MOVL C00664 V=800.0 PL=0
MOVL C00665 V=800.0 PL=0
MOVL C00666 V=800.0 PL=0
MOVL C00667 V=800.0 PL=0
MOVL C00668 V=800.0 PL=0
MOVL C00669 V=800.0 PL=0
MOVL C00670 V=800.0 PL=0
MOVL C00671 V=800.0 PL=0
MOVL C00672 V=800.0 PL=0
MOVL C00673 V=800.0 PL=0
MOVL C00674 V=800.0 PL=0
MOVL C00675 V=800.0 PL=0
MOVL C00676 V=800.0 PL=0
MOVL C00677 V=800.0 PL=0
MOVL C00678 V=800.0 PL=0
MOVL C00679 V=800.0 PL=0
MOVL C00680 V=800.0 PL=0
MOVL C00681 V=800.0 PL=0
MOVL C00682 V=800.0 PL=0
MOVL C00683 V=800.0 PL=0
MOVL C00684 V=800.0 PL=0
MOVL C00685 V=800.0 PL=0
MOVL C00686 V=800.0 PL=0
MOVL C00687 V=800.0 PL=0
MOVL C00688 V=800.0 PL=0
MOVL C00689 V=800.0 PL=0
MOVL C00690 V=800.0 PL=0
MOVL C00691 V=800.0 PL=0
MOVL C00692 V=800.0 PL=0
MOVL C00693 V=800.0 PL=0
MOVL C00694 V=800.0 PL=0
MOVL C00695 V=800.0 PL=0
MOVL C00696 V=800.0 PL=0
MOVL C00697 V=800.0 PL=0
MOVL C00698 V=800.0 PL=0
MOVL C00699 V=800.0 PL=0
MOVL C00700 V=800.0 PL=0
MOVL C00701 V=800.0 PL=0
MOVL C00702 V=800.0 PL=0
MOVL C00703 V=800.0 PL=0
MOVL C00704 V=800.0 PL=0
MOVL C00705 V=800.0 PL=0
MOVL C00706 V=800.0 PL=0
MOVL C00707 V=800.0 PL=0
MOVL C00708 V=800.0 PL=0
MOVL C00709 V=800.0 PL=0
MOVL C00710 V=800.0 PL=0
MOVL C00711 V=800.0 PL=0
MOVL C00712 V=800.0 PL=0
MOVL C00713 V=800.0 PL=0
MOVL C00714 V=800.0 PL=0
MOVL C00715 V=800.0 PL=0
MOVL C00716 V=800.0 PL=0
MOVL C00717 V=800.0 PL=0
MOVL C00718 V=800.0 PL=0
MOVL C00719 V=800.0 PL=0
MOVL C00720 V=800.0 PL=0
MOVL C00721 V=800.0 PL=0
MOVL C00722 V=800.0 PL=0
MOVL C00723 V=800.0 PL=0
MOVL C00724 V=800.0 PL=0
MOVL C00725 V=800.0 PL=0
MOVL C00726 V=800.0 PL=0
MOVL C00727 V=800.0 PL=0
MOVL C00728 V=800.0 PL=0
MOVL C00729 V=800.0 PL=0
MOVL C00730 V=800.0 PL=0
MOVL C00731 V=800.0 PL=0
MOVL C00732 V=800.0 PL=0
MOVL C00733 V=800.0 PL=0
MOVL C00734 V=800.0 PL=0
MOVL C00735 V=800.0 PL=0
MOVL C00736 V=800.0 PL=0
MOVL C00737 V=800.0 PL=0
MOVL C00738 V=800.0 PL=0
MOVL C00739 V=800.0 PL=0
MOVL C00740 V=800.0 PL=0
MOVL C00741 V=800.0 PL=0
MOVL C00742 V=800.0 PL=0
MOVL C00743 V=800.0 PL=0
MOVL C00744 V=800.0 PL=0
MOVL C00745 V=800.0 PL=0
MOVL C00746 V=800.0 PL=0
MOVL C00747 V=800.0 PL=0
MOVL C00748 V=800.0 PL=0
MOVL C00749 V=800.0 PL=0
MOVL C00750 V=800.0 PL=0
MOVL C00751 V=800.0 PL=0
MOVL C00752 V=800.0 PL=0
MOVL C00753 V=800.0 PL=0
MOVL C00754 V=800.0 PL=0
MOVL C00755 V=800.0 PL=0
MOVL C00756 V=800.0 PL=0
MOVL C00757 V=800.0 PL=0
MOVL C00758 V=800.0 PL=0
MOVL C00759 V=800.0 PL=0
MOVL C00760 V=800.0 PL=0
MOVL C00761 V=800.0 PL=0
MOVL C00762 V=800.0 PL=0
MOVL C00763 V=800.0 PL=0
MOVL C00764 V=800.0 PL=0
MOVL C00765 V=800.0 PL=0
MOVL C00766 V=800.0 PL=0
MOVL C00767 V=800.0 PL=0
MOVL C00768 V=800.0 PL=0
MOVL C00769 V=800.0 PL=0
MOVL C00770 V=800.0 PL=0
MOVL C00771 V=800.0 PL=0
MOVL C00772 V=800.0 PL=0
MOVL C00773 V=800.0 PL=0
MOVL C00774 V=800.0 PL=0
MOVL C00775 V=800.0 PL=0
MOVL C00776 V=800.0 PL=0
MOVL C00777 V=800.0 PL=0
MOVL C00778 V=800.0 PL=0
MOVL C00779 V=800.0 PL=0
MOVL C00780 V=800.0 PL=0
MOVL C00781 V=800.0 PL=0
MOVL C00782 V=800.0 PL=0
MOVL C00783 V=800.0 PL=0
MOVL C00784 V=800.0 PL=0
MOVL C00785 V=800.0 PL=0
MOVL C00786 V=800.0 PL=0
MOVL C00787 V=800.0 PL=0
MOVL C00788 V=800.0 PL=0
MOVL C00789 V=800.0 PL=0
MOVL C00790 V=800.0 PL=0
MOVL C00791 V=800.0 PL=0
MOVL C00792 V=800.0 PL=0
MOVL C00793 V=800.0 PL=0
MOVL C00794 V=800.0 PL=0
MOVL C00795 V=800.0 PL=0
MOVL C00796 V=800.0 PL=0
MOVL C00797 V=800.0 PL=0
MOVL C00798 V=800.0 PL=0
MOVL C00799 V=800.0 PL=0
MOVL C00800 V=800.0 PL=0
MOVL C00801 V=800.0 PL=0
MOVL C00802 V=800.0 PL=0
MOVL C00803 V=800.0 PL=0
MOVL C00804 V=800.0 PL=0
MOVL C00805 V=800.0 PL=0
MOVL C00806 V=800.0 PL=0
MOVL C00807 V=800.0 PL=0
MOVL C00808 V=800.0 PL=0
MOVL C00809 V=800.0 PL=0
MOVL C00810 V=800.0 PL=0
MOVL C00811 V=800.0 PL=0
MOVL C00812 V=800.0 PL=0
MOVL C00813 V=800.0 PL=0
MOVL C00814 V=800.0 PL=0
MOVL C00815 V=800.0 PL=0
MOVL C00816 V=800.0 PL=0
MOVL C00817 V=800.0 PL=0
MOVL C00818 V=800.0 PL=0
MOVL C00819 V=800.0 PL=0
MOVL C00820 V=800.0 PL=0
MOVL C00821 V=800.0 PL=0
MOVL C00822 V=800.0 PL=0
MOVL C00823 V=800.0 PL=0
MOVL C00824 V=800.0 PL=0
MOVL C00825 V=800.0 PL=0
MOVL C00826 V=800.0 PL=0
MOVL C00827 V=800.0 PL=0
MOVL C00828 V=800.0 PL=0
MOVL C00829 V=800.0 PL=0
MOVL C00830 V=800.0 PL=0
MOVL C00831 V=800.0 PL=0
MOVL C00832 V=800.0 PL=0
MOVL C00833 V=800.0 PL=0
MOVL C00834 V=800.0 PL=0
MOVL C00835 V=800.0 PL=0
MOVL C00836 V=800.0 PL=0
MOVL C00837 V=800.0 PL=0
MOVL C00838 V=800.0 PL=0
MOVL C00839 V=800.0 PL=0
MOVL C00840 V=800.0 PL=0
MOVL C00841 V=800.0 PL=0
MOVL C00842 V=800.0 PL=0
MOVL C00843 V=800.0 PL=0
MOVL C00844 V=800.0 PL=0
MOVL C00845 V=800.0 PL=0
MOVL C00846 V=800.0 PL=0
MOVL C00847 V=800.0 PL=0
MOVL C00848 V=800.0 PL=0
MOVL C00849 V=800.0 PL=0
MOVL C00850 V=800.0 PL=0
MOVL C00851 V=800.0 PL=0
MOVL C00852 V=800.0 PL=0
MOVL C00853 V=800.0 PL=0
MOVL C00854 V=800.0 PL=0
MOVL C00855 V=800.0 PL=0
MOVL C00856 V=800.0 PL=0
MOVL C00857 V=800.0 PL=0
MOVL C00858 V=800.0 PL=0
MOVL C00859 V=800.0 PL=0
MOVL C00860 V=800.0 PL=0
MOVL C00861 V=800.0 PL=0
MOVL C00862 V=800.0 PL=0
MOVL C00863 V=800.0 PL=0
MOVL C00864 V=800.0 PL=0
MOVL C00865 V=800.0 PL=0
MOVL C00866 V=800.0 PL=0
MOVL C00867 V=800.0 PL=0
MOVL C00868 V=800.0 PL=0
MOVL C00869 V=800.0 PL=0
MOVL C00870 V=800.0 PL=0
MOVL C00871 V=800.0 PL=0
MOVL C00872 V=800.0 PL=0
MOVL C00873 V=800.0 PL=0
MOVL C00874 V=800.0 PL=0
MOVL C00875 V=800.0 PL=0
MOVL C00876 V=800.0 PL=0
MOVL C00877 V=800.0 PL=0
MOVL C00878 V=800.0 PL=0
MOVL C00879 V=800.0 PL=0
MOVL C00880 V=800.0 PL=0
MOVL C00881 V=800.0 PL=0
MOVL C00882 V=800.0 PL=0
MOVL C00883 V=800.0 PL=0
MOVL C00884 V=800.0 PL=0
MOVL C00885 V=800.0 PL=0
MOVL C00886 V=800.0 PL=0
MOVL C00887 V=800.0 PL=0
MOVL C00888 V=800.0 PL=0
MOVL C00889 V=800.0 PL=0
MOVL C00890 V=800.0 PL=0
MOVL C00891 V=800.0 PL=0
MOVL C00892 V=800.0 PL=0
MOVL C00893 V=800.0 PL=0
MOVL C00894 V=800.0 PL=0
MOVL C00895 V=800.0 PL=0
MOVL C00896 V=800.0 PL=0
MOVL C00897 V=800.0 PL=0
MOVL C00898 V=800.0 PL=0
MOVL C00899 V=800.0 PL=0
MOVL C00900 V=800.0 PL=0
MOVL C00901 V=800.0 PL=0
MOVL C00902 V=800.0 PL=0
MOVL C00903 V=800.0 PL=0
MOVL C00904 V=800.0 PL=0
MOVL C00905 V=800.0 PL=0
MOVL C00906 V=800.0 PL=0
MOVL C00907 V=800.0 PL=0
MOVL C00908 V=800.0 PL=0
MOVL C00909 V=800.0 PL=0
MOVL C00910 V=800.0 PL=0
MOVL C00911 V=800.0 PL=0
MOVL C00912 V=800.0 PL=0
MOVL C00913 V=800.0 PL=0
MOVL C00914 V=800.0 PL=0
MOVL C00915 V=800.0 PL=0
MOVL C00916 V=800.0 PL=0
MOVL C00917 V=800.0 PL=0
MOVL C00918 V=800.0 PL=0
MOVL C00919 V=800.0 PL=0
MOVL C00920 V=800.0 PL=0
MOVL C00921 V=800.0 PL=0
MOVL C00922 V=800.0 PL=0
MOVL C00923 V=800.0 PL=0
MOVL C00924 V=800.0 PL=0
MOVL C00925 V=800.0 PL=0
MOVL C00926 V=800.0 PL=0
MOVL C00927 V=800.0 PL=0
MOVL C00928 V=800.0 PL=0
MOVL C00929 V=800.0 PL=0
MOVL C00930 V=800.0 PL=0
MOVL C00931 V=800.0 PL=0
MOVL C00932 V=800.0 PL=0
MOVL C00933 V=800.0 PL=0
MOVL C00934 V=800.0 PL=0
MOVL C00935 V=800.0 PL=0
MOVL C00936 V=800.0 PL=0
MOVL C00937 V=800.0 PL=0
MOVL C00938 V=800.0 PL=0
MOVL C00939 V=800.0 PL=0
MOVL C00940 V=800.0 PL=0
MOVL C00941 V=800.0 PL=0
MOVL C00942 V=800.0 PL=0
MOVL C00943 V=800.0 PL=0
MOVL C00944 V=800.0 PL=0
MOVL C00945 V=800.0 PL=0
MOVL C00946 V=800.0 PL=0
MOVL C00947 V=800.0 PL=0
MOVL C00948 V=800.0 PL=0
MOVL C00949 V=800.0 PL=0
MOVL C00950 V=800.0 PL=0
MOVL C00951 V=800.0 PL=0
MOVL C00952 V=800.0 PL=0
MOVL C00953 V=800.0 PL=0
MOVL C00954 V=800.0 PL=0
MOVL C00955 V=800.0 PL=0
MOVL C00956 V=800.0 PL=0
MOVL C00957 V=800.0 PL=0
MOVL C00958 V=800.0 PL=0
MOVL C00959 V=800.0 PL=0
MOVL C00960 V=800.0 PL=0
MOVL C00961 V=800.0 PL=0
MOVL C00962 V=800.0 PL=0
MOVL C00963 V=800.0 PL=0
MOVL C00964 V=800.0 PL=0
MOVL C00965 V=800.0 PL=0
MOVL C00966 V=800.0 PL=0
MOVL C00967 V=800.0 PL=0
MOVL C00968 V=800.0 PL=0
MOVL C00969 V=800.0 PL=0
MOVL C00970 V=800.0 PL=0
MOVL C00971 V=800.0 PL=0
MOVL C00972 V=800.0 PL=0
MOVL C00973 V=800.0 PL=0
MOVL C00974 V=800.0 PL=0
MOVL C00975 V=800.0 PL=0
MOVL C00976 V=800.0 PL=0
MOVL C00977 V=800.0 PL=0
MOVL C00978 V=800.0 PL=0
MOVL C00979 V=800.0 PL=0
MOVL C00980 V=800.0 PL=0
MOVL C00981 V=800.0 PL=0
MOVL C00982 V=800.0 PL=0
MOVL C00983 V=800.0 PL=0
MOVL C00984 V=800.0 PL=0
MOVL C00985 V=800.0 PL=0
MOVL C00986 V=800.0 PL=0
MOVL C00987 V=800.0 PL=0
MOVL C00988 V=800.0 PL=0
MOVL C00989 V=800.0 PL=0
MOVL C00990 V=800.0 PL=0
MOVL C00991 V=800.0 PL=0
MOVL C00992 V=800.0 PL=0
MOVL C00993 V=800.0 PL=0
MOVL C00994 V=800.0 PL=0
MOVL C00995 V=800.0 PL=0
MOVL C00996 V=800.0 PL=0
MOVL C00997 V=800.0 PL=0
MOVL C00998 V=800.0 PL=0
MOVL C00999 V=800.0 PL=0
MOVL C01000 V=800.0 PL=0
MOVL C01001 V=800.0 PL=0
MOVL C01002 V=800.0 PL=0
MOVL C01003 V=800.0 PL=0
MOVL C01004 V=800.0 PL=0
MOVL C01005 V=800.0 PL=0
MOVL C01006 V=800.0 PL=0
MOVL C01007 V=800.0 PL=0
MOVL C01008 V=800.0 PL=0
MOVL C01009 V=800.0 PL=0
MOVL C01010 V=800.0 PL=0
MOVL C01011 V=800.0 PL=0
MOVL C01012 V=800.0 PL=0
MOVL C01013 V=800.0 PL=0
MOVL C01014 V=800.0 PL=0
MOVL C01015 V=800.0 PL=0
MOVL C01016 V=800.0 PL=0
MOVL C01017 V=800.0 PL=0
MOVL C01018 V=800.0 PL=0
MOVL C01019 V=800.0 PL=0
MOVL C01020 V=800.0 PL=0
MOVL C01021 V=800.0 PL=0
MOVL C01022 V=800.0 PL=0
MOVL C01023 V=800.0 PL=0
MOVL C01024 V=800.0 PL=0
MOVL C01025 V=800.0 PL=0
MOVL C01026 V=800.0 PL=0
MOVL C01027 V=800.0 PL=0
MOVL C01028 V=800.0 PL=0
MOVL C01029 V=800.0 PL=0
MOVL C01030 V=800.0 PL=0
MOVL C01031 V=800.0 PL=0
MOVL C01032 V=800.0 PL=0
MOVL C01033 V=800.0 PL=0
MOVL C01034 V=800.0 PL=0
MOVL C01035 V=800.0 PL=0
MOVL C01036 V=800.0 PL=0
MOVL C01037 V=800.0 PL=0
MOVL C01038 V=800.0 PL=0
MOVL C01039 V=800.0 PL=0
MOVL C01040 V=800.0 PL=0
MOVL C01041 V=800.0 PL=0
MOVL C01042 V=800.0 PL=0
MOVL C01043 V=800.0 PL=0
MOVL C01044 V=800.0 PL=0
MOVL C01045 V=800.0 PL=0
MOVL C01046 V=800.0 PL=0
MOVL C01047 V=800.0 PL=0
MOVL C01048 V=800.0 PL=0
MOVL C01049 V=800.0 PL=0
MOVL C01050 V=800.0 PL=0
MOVL C01051 V=800.0 PL=0
MOVL C01052 V=800.0 PL=0
MOVL C01053 V=800.0 PL=0
MOVL C01054 V=800.0 PL=0
MOVL C01055 V=800.0 PL=0
MOVL C01056 V=800.0 PL=0
MOVL C01057 V=800.0 PL=0
MOVL C01058 V=800.0 PL=0
MOVL C01059 V=800.0 PL=0
MOVL C01060 V=800.0 PL=0
MOVL C01061 V=800.0 PL=0
MOVL C01062 V=800.0 PL=0
MOVL C01063 V=800.0 PL=0
MOVL C01064 V=800.0 PL=0
MOVL C01065 V=800.0 PL=0
MOVL C01066 V=800.0 PL=0
MOVL C01067 V=800.0 PL=0
MOVL C01068 V=800.0 PL=0
MOVL C01069 V=800.0 PL=0
MOVL C01070 V=800.0 PL=0
MOVL C01071 V=800.0 PL=0
MOVL C01072 V=800.0 PL=0
MOVL C01073 V=800.0 PL=0
MOVL C01074 V=800.0 PL=0
MOVL C01075 V=800.0 PL=0
MOVL C01076 V=800.0 PL=0
MOVL C01077 V=800.0 PL=0
MOVL C01078 V=800.0 PL=0
MOVL C01079 V=800.0 PL=0
MOVL C01080 V=800.0 PL=0
MOVL C01081 V=800.0 PL=0
MOVL C01082 V=800.0 PL=0
MOVL C01083 V=800.0 PL=0
MOVL C01084 V=800.0 PL=0
MOVL C01085 V=800.0 PL=0
MOVL C01086 V=800.0 PL=0
MOVL C01087 V=800.0 PL=0
MOVL C01088 V=800.0 PL=0
MOVL C01089 V=800.0 PL=0
MOVL C01090 V=800.0 PL=0
MOVL C01091 V=800.0 PL=0
MOVL C01092 V=800.0 PL=0
MOVL C01093 V=800.0 PL=0
MOVL C01094 V=800.0 PL=0
MOVL C01095 V=800.0 PL=0
MOVL C01096 V=800.0 PL=0
MOVL C01097 V=800.0 PL=0
MOVL C01098 V=800.0 PL=0
MOVL C01099 V=800.0 PL=0
MOVL C01100 V=800.0 PL=0
MOVL C01101 V=800.0 PL=0
MOVL C01102 V=800.0 PL=0
MOVL C01103 V=800.0 PL=0
MOVL C01104 V=800.0 PL=0
MOVL C01105 V=800.0 PL=0
MOVL C01106 V=800.0 PL=0
MOVL C01107 V=800.0 PL=0
MOVL C01108 V=800.0 PL=0
MOVL C01109 V=800.0 PL=0
MOVL C01110 V=800.0 PL=0
MOVL C01111 V=800.0 PL=0
MOVL C01112 V=800.0 PL=0
MOVL C01113 V=800.0 PL=0
MOVL C01114 V=800.0 PL=0
MOVL C01115 V=800.0 PL=0
MOVL C01116 V=800.0 PL=0
MOVL C01117 V=800.0 PL=0
MOVL C01118 V=800.0 PL=0
MOVL C01119 V=800.0 PL=0
MOVL C01120 V=800.0 PL=0
MOVL C01121 V=800.0 PL=0
MOVL C01122 V=800.0 PL=0
MOVL C01123 V=800.0 PL=0
MOVL C01124 V=800.0 PL=0
MOVL C01125 V=800.0 PL=0
MOVL C01126 V=800.0 PL=0
MOVL C01127 V=800.0 PL=0
MOVL C01128 V=800.0 PL=0
MOVL C01129 V=800.0 PL=0
MOVL C01130 V=800.0 PL=0
MOVL C01131 V=800.0 PL=0
MOVL C01132 V=800.0 PL=0
MOVL C01133 V=800.0 PL=0
MOVL C01134 V=800.0 PL=0
MOVL C01135 V=800.0 PL=0
MOVL C01136 V=800.0 PL=0
MOVL C01137 V=800.0 PL=0
MOVL C01138 V=800.0 PL=0
MOVL C01139 V=800.0 PL=0
MOVL C01140 V=800.0 PL=0
MOVL C01141 V=800.0 PL=0
MOVL C01142 V=800.0 PL=0
MOVL C01143 V=800.0 PL=0
MOVL C01144 V=800.0 PL=0
MOVL C01145 V=800.0 PL=0
MOVL C01146 V=800.0 PL=0
MOVL C01147 V=800.0 PL=0
MOVL C01148 V=800.0 PL=0
MOVL C01149 V=800.0 PL=0
MOVL C01150 V=800.0 PL=0
MOVL C01151 V=800.0 PL=0
MOVL C01152 V=800.0 PL=0
MOVL C01153 V=800.0 PL=0
MOVL C01154 V=800.0 PL=0
MOVL C01155 V=800.0 PL=0
MOVL C01156 V=800.0 PL=0
MOVL C01157 V=800.0 PL=0
MOVL C01158 V=800.0 PL=0
MOVL C01159 V=800.0 PL=0
MOVL C01160 V=800.0 PL=0
MOVL C01161 V=800.0 PL=0
MOVL C01162 V=800.0 PL=0
MOVL C01163 V=800.0 PL=0
MOVL C01164 V=800.0 PL=0
MOVL C01165 V=800.0 PL=0
MOVL C01166 V=800.0 PL=0
MOVL C01167 V=800.0 PL=0
MOVL C01168 V=800.0 PL=0
MOVL C01169 V=800.0 PL=0
MOVL C01170 V=800.0 PL=0
MOVL C01171 V=800.0 PL=0
MOVL C01172 V=800.0 PL=0
MOVL C01173 V=800.0 PL=0
MOVL C01174 V=800.0 PL=0
MOVL C01175 V=800.0 PL=0
MOVL C01176 V=800.0 PL=0
MOVL C01177 V=800.0 PL=0
MOVL C01178 V=800.0 PL=0
MOVL C01179 V=800.0 PL=0
MOVL C01180 V=800.0 PL=0
MOVL C01181 V=800.0 PL=0
MOVL C01182 V=800.0 PL=0
MOVL C01183 V=800.0 PL=0
MOVL C01184 V=800.0 PL=0
MOVL C01185 V=800.0 PL=0
MOVL C01186 V=800.0 PL=0
MOVL C01187 V=800.0 PL=0
MOVL C01188 V=800.0 PL=0
MOVL C01189 V=800.0 PL=0
MOVL C01190 V=800.0 PL=0
MOVL C01191 V=800.0 PL=0
MOVL C01192 V=800.0 PL=0
MOVL C01193 V=800.0 PL=0
MOVL C01194 V=800.0 PL=0
MOVL C01195 V=800.0 PL=0
MOVL C01196 V=800.0 PL=0
MOVL C01197 V=800.0 PL=0
MOVL C01198 V=800.0 PL=0
MOVL C01199 V=800.0 PL=0
MOVL C01200 V=800.0 PL=0
MOVL C01201 V=800.0 PL=0
MOVL C01202 V=800.0 PL=0
MOVL C01203 V=800.0 PL=0
MOVL C01204 V=800.0 PL=0
MOVL C01205 V=800.0 PL=0
MOVL C01206 V=800.0 PL=0
MOVL C01207 V=800.0 PL=0
MOVL C01208 V=800.0 PL=0
MOVL C01209 V=800.0 PL=0
MOVL C01210 V=800.0 PL=0
MOVL C01211 V=800.0 PL=0
MOVL C01212 V=800.0 PL=0
MOVL C01213 V=800.0 PL=0
MOVL C01214 V=800.0 PL=0
MOVL C01215 V=800.0 PL=0
MOVL C01216 V=800.0 PL=0
MOVL C01217 V=800.0 PL=0
MOVL C01218 V=800.0 PL=0
MOVL C01219 V=800.0 PL=0
MOVL C01220 V=800.0 PL=0
MOVL C01221 V=800.0 PL=0
MOVL C01222 V=800.0 PL=0
MOVL C01223 V=800.0 PL=0
MOVL C01224 V=800.0 PL=0
MOVL C01225 V=800.0 PL=0
MOVL C01226 V=800.0 PL=0
MOVL C01227 V=800.0 PL=0
MOVL C01228 V=800.0 PL=0
MOVL C01229 V=800.0 PL=0
MOVL C01230 V=800.0 PL=0
MOVL C01231 V=800.0 PL=0
MOVL C01232 V=800.0 PL=0
MOVL C01233 V=800.0 PL=0
MOVL C01234 V=800.0 PL=0
MOVL C01235 V=800.0 PL=0
MOVL C01236 V=800.0 PL=0
MOVL C01237 V=800.0 PL=0
MOVL C01238 V=800.0 PL=0
MOVL C01239 V=800.0 PL=0
MOVL C01240 V=800.0 PL=0
MOVL C01241 V=800.0 PL=0
MOVL C01242 V=800.0 PL=0
MOVL C01243 V=800.0 PL=0
MOVL C01244 V=800.0 PL=0
MOVL C01245 V=800.0 PL=0
MOVL C01246 V=800.0 PL=0
MOVL C01247 V=800.0 PL=0
MOVL C01248 V=800.0 PL=0
MOVL C01249 V=800.0 PL=0
MOVL C01250 V=800.0 PL=0
MOVL C01251 V=800.0 PL=0
MOVL C01252 V=800.0 PL=0
MOVL C01253 V=800.0 PL=0
MOVL C01254 V=800.0 PL=0
MOVL C01255 V=800.0 PL=0
MOVL C01256 V=800.0 PL=0
MOVL C01257 V=800.0 PL=0
MOVL C01258 V=800.0 PL=0
MOVL C01259 V=800.0 PL=0
MOVL C01260 V=800.0 PL=0
MOVL C01261 V=800.0 PL=0
MOVL C01262 V=800.0 PL=0
MOVL C01263 V=800.0 PL=0
MOVL C01264 V=800.0 PL=0
MOVL C01265 V=800.0 PL=0
MOVL C01266 V=800.0 PL=0
MOVL C01267 V=800.0 PL=0
MOVL C01268 V=800.0 PL=0
MOVL C01269 V=800.0 PL=0
MOVL C01270 V=800.0 PL=0
MOVL C01271 V=800.0 PL=0
MOVL C01272 V=800.0 PL=0
MOVL C01273 V=800.0 PL=0
MOVL C01274 V=800.0 PL=0
MOVL C01275 V=800.0 PL=0
MOVL C01276 V=800.0 PL=0
MOVL C01277 V=800.0 PL=0
MOVL C01278 V=800.0 PL=0
MOVL C01279 V=800.0 PL=0
MOVL C01280 V=800.0 PL=0
MOVL C01281 V=800.0 PL=0
MOVL C01282 V=800.0 PL=0
MOVL C01283 V=800.0 PL=0
MOVL C01284 V=800.0 PL=0
MOVL C01285 V=800.0 PL=0
MOVL C01286 V=800.0 PL=0
MOVL C01287 V=800.0 PL=0
MOVL C01288 V=800.0 PL=0
MOVL C01289 V=800.0 PL=0
MOVL C01290 V=800.0 PL=0
MOVL C01291 V=800.0 PL=0
MOVL C01292 V=800.0 PL=0
MOVL C01293 V=800.0 PL=0
MOVL C01294 V=800.0 PL=0
MOVL C01295 V=800.0 PL=0
MOVL C01296 V=800.0 PL=0
MOVL C01297 V=800.0 PL=0
MOVL C01298 V=800.0 PL=0
MOVL C01299 V=800.0 PL=0
MOVL C01300 V=800.0 PL=0
MOVL C01301 V=800.0 PL=0
MOVL C01302 V=800.0 PL=0
MOVL C01303 V=800.0 PL=0
MOVL C01304 V=800.0 PL=0
MOVL C01305 V=800.0 PL=0
MOVL C01306 V=800.0 PL=0
MOVL C01307 V=800.0 PL=0
MOVL C01308 V=800.0 PL=0
MOVL C01309 V=800.0 PL=0
MOVL C01310 V=800.0 PL=0
MOVL C01311 V=800.0 PL=0
MOVL C01312 V=800.0 PL=0
MOVL C01313 V=800.0 PL=0
MOVL C01314 V=800.0 PL=0
MOVL C01315 V=800.0 PL=0
MOVL C01316 V=800.0 PL=0
MOVL C01317 V=800.0 PL=0
MOVL C01318 V=800.0 PL=0
MOVL C01319 V=800.0 PL=0
MOVL C01320 V=800.0 PL=0
MOVL C01321 V=800.0 PL=0
MOVL C01322 V=800.0 PL=0
MOVL C01323 V=800.0 PL=0
MOVL C01324 V=800.0 PL=0
MOVL C01325 V=800.0 PL=0
MOVL C01326 V=800.0 PL=0
MOVL C01327 V=800.0 PL=0
MOVL C01328 V=800.0 PL=0
MOVL C01329 V=800.0 PL=0
MOVL C01330 V=800.0 PL=0
MOVL C01331 V=800.0 PL=0
MOVL C01332 V=800.0 PL=0
MOVL C01333 V=800.0 PL=0
MOVL C01334 V=800.0 PL=0
MOVL C01335 V=800.0 PL=0
MOVL C01336 V=800.0 PL=0
MOVL C01337 V=800.0 PL=0
MOVL C01338 V=800.0 PL=0
MOVL C01339 V=800.0 PL=0
MOVL C01340 V=800.0 PL=0
MOVL C01341 V=800.0 PL=0
MOVL C01342 V=800.0 PL=0
MOVL C01343 V=800.0 PL=0
MOVL C01344 V=800.0 PL=0
MOVL C01345 V=800.0 PL=0
MOVL C01346 V=800.0 PL=0
MOVL C01347 V=800.0 PL=0
MOVL C01348 V=800.0 PL=0
MOVL C01349 V=800.0 PL=0
MOVL C01350 V=800.0 PL=0
MOVL C01351 V=800.0 PL=0
MOVL C01352 V=800.0 PL=0
MOVL C01353 V=800.0 PL=0
MOVL C01354 V=800.0 PL=0
MOVL C01355 V=800.0 PL=0
MOVL C01356 V=800.0 PL=0
MOVL C01357 V=800.0 PL=0
MOVL C01358 V=800.0 PL=0
MOVL C01359 V=800.0 PL=0
MOVL C01360 V=800.0 PL=0
MOVL C01361 V=800.0 PL=0
MOVL C01362 V=800.0 PL=0
MOVL C01363 V=800.0 PL=0
MOVL C01364 V=800.0 PL=0
MOVL C01365 V=800.0 PL=0
MOVL C01366 V=800.0 PL=0
MOVL C01367 V=800.0 PL=0
MOVL C01368 V=800.0 PL=0
MOVL C01369 V=800.0 PL=0
MOVL C01370 V=800.0 PL=0
MOVL C01371 V=800.0 PL=0
MOVL C01372 V=800.0 PL=0
MOVL C01373 V=800.0 PL=0
MOVL C01374 V=800.0 PL=0
MOVL C01375 V=800.0 PL=0
MOVL C01376 V=800.0 PL=0
MOVL C01377 V=800.0 PL=0
MOVL C01378 V=800.0 PL=0
MOVL C01379 V=800.0 PL=0
MOVL C01380 V=800.0 PL=0
MOVL C01381 V=800.0 PL=0
MOVL C01382 V=800.0 PL=0
MOVL C01383 V=800.0 PL=0
MOVL C01384 V=800.0 PL=0
MOVL C01385 V=800.0 PL=0
MOVL C01386 V=800.0 PL=0
MOVL C01387 V=800.0 PL=0
MOVL C01388 V=800.0 PL=0
MOVL C01389 V=800.0 PL=0
MOVL C01390 V=800.0 PL=0
MOVL C01391 V=800.0 PL=0
MOVL C01392 V=800.0 PL=0
MOVL C01393 V=800.0 PL=0
MOVL C01394 V=800.0 PL=0
MOVL C01395 V=800.0 PL=0
MOVL C01396 V=800.0 PL=0
MOVL C01397 V=800.0 PL=0
MOVL C01398 V=800.0 PL=0
MOVL C01399 V=800.0 PL=0
MOVL C01400 V=800.0 PL=0
MOVL C01401 V=800.0 PL=0
MOVL C01402 V=800.0 PL=0
MOVL C01403 V=800.0 PL=0
MOVL C01404 V=800.0 PL=0
MOVL C01405 V=800.0 PL=0
MOVL C01406 V=800.0 PL=0
MOVL C01407 V=800.0 PL=0
MOVL C01408 V=800.0 PL=0
MOVL C01409 V=800.0 PL=0
MOVL C01410 V=800.0 PL=0
MOVL C01411 V=800.0 PL=0
MOVL C01412 V=800.0 PL=0
MOVL C01413 V=800.0 PL=0
MOVL C01414 V=800.0 PL=0
MOVL C01415 V=800.0 PL=0
MOVL C01416 V=800.0 PL=0
MOVL C01417 V=800.0 PL=0
MOVL C01418 V=800.0 PL=0
MOVL C01419 V=800.0 PL=0
MOVL C01420 V=800.0 PL=0
MOVL C01421 V=800.0 PL=0
MOVL C01422 V=800.0 PL=0
MOVL C01423 V=800.0 PL=0
MOVL C01424 V=800.0 PL=0
MOVL C01425 V=800.0 PL=0
MOVL C01426 V=800.0 PL=0
MOVL C01427 V=800.0 PL=0
MOVL C01428 V=800.0 PL=0
MOVL C01429 V=800.0 PL=0
MOVL C01430 V=800.0 PL=0
MOVL C01431 V=800.0 PL=0
MOVL C01432 V=800.0 PL=0
MOVL C01433 V=800.0 PL=0
MOVL C01434 V=800.0 PL=0
MOVL C01435 V=800.0 PL=0
MOVL C01436 V=800.0 PL=0
MOVL C01437 V=800.0 PL=0
MOVL C01438 V=800.0 PL=0
MOVL C01439 V=800.0 PL=0
MOVL C01440 V=800.0 PL=0
MOVL C01441 V=800.0 PL=0
MOVL C01442 V=800.0 PL=0
MOVL C01443 V=800.0 PL=0
MOVL C01444 V=800.0 PL=0
MOVL C01445 V=800.0 PL=0
MOVL C01446 V=800.0 PL=0
MOVL C01447 V=800.0 PL=0
MOVL C01448 V=800.0 PL=0
MOVL C01449 V=800.0 PL=0
MOVL C01450 V=800.0 PL=0
MOVL C01451 V=800.0 PL=0
MOVL C01452 V=800.0 PL=0
MOVL C01453 V=800.0 PL=0
MOVL C01454 V=800.0 PL=0
MOVL C01455 V=800.0 PL=0
MOVL C01456 V=800.0 PL=0
MOVL C01457 V=800.0 PL=0
MOVL C01458 V=800.0 PL=0
MOVL C01459 V=800.0 PL=0
MOVL C01460 V=800.0 PL=0
MOVL C01461 V=800.0 PL=0
MOVL C01462 V=800.0 PL=0
MOVL C01463 V=800.0 PL=0
MOVL C01464 V=800.0 PL=0
MOVL C01465 V=800.0 PL=0
MOVL C01466 V=800.0 PL=0
MOVL C01467 V=800.0 PL=0
MOVL C01468 V=800.0 PL=0
MOVL C01469 V=800.0 PL=0
MOVL C01470 V=800.0 PL=0
MOVL C01471 V=800.0 PL=0
MOVL C01472 V=800.0 PL=0
MOVL C01473 V=800.0 PL=0
MOVL C01474 V=800.0 PL=0
MOVL C01475 V=800.0 PL=0
MOVL C01476 V=800.0 PL=0
MOVL C01477 V=800.0 PL=0
MOVL C01478 V=800.0 PL=0
MOVL C01479 V=800.0 PL=0
MOVL C01480 V=800.0 PL=0
MOVL C01481 V=800.0 PL=0
MOVL C01482 V=800.0 PL=0
MOVL C01483 V=800.0 PL=0
MOVL C01484 V=800.0 PL=0
MOVL C01485 V=800.0 PL=0
MOVL C01486 V=800.0 PL=0
MOVL C01487 V=800.0 PL=0
MOVL C01488 V=800.0 PL=0
MOVL C01489 V=800.0 PL=0
MOVL C01490 V=800.0 PL=0
MOVL C01491 V=800.0 PL=0
MOVL C01492 V=800.0 PL=0
MOVL C01493 V=800.0 PL=0
MOVL C01494 V=800.0 PL=0
MOVL C01495 V=800.0 PL=0
MOVL C01496 V=800.0 PL=0
MOVL C01497 V=800.0 PL=0
MOVL C01498 V=800.0 PL=0
MOVL C01499 V=800.0 PL=0
MOVL C01500 V=800.0 PL=0
MOVL C01501 V=800.0 PL=0
MOVL C01502 V=800.0 PL=0
MOVL C01503 V=800.0 PL=0
MOVL C01504 V=800.0 PL=0
MOVL C01505 V=800.0 PL=0
MOVL C01506 V=800.0 PL=0
MOVL C01507 V=800.0 PL=0
MOVL C01508 V=800.0 PL=0
MOVL C01509 V=800.0 PL=0
MOVL C01510 V=800.0 PL=0
MOVL C01511 V=800.0 PL=0
MOVL C01512 V=800.0 PL=0
MOVL C01513 V=800.0 PL=0
MOVL C01514 V=800.0 PL=0
MOVL C01515 V=800.0 PL=0
MOVL C01516 V=800.0 PL=0
MOVL C01517 V=800.0 PL=0
MOVL C01518 V=800.0 PL=0
MOVL C01519 V=800.0 PL=0
MOVL C01520 V=800.0 PL=0
MOVL C01521 V=800.0 PL=0
MOVL C01522 V=800.0 PL=0
MOVL C01523 V=800.0 PL=0
MOVL C01524 V=800.0 PL=0
MOVL C01525 V=800.0 PL=0
MOVL C01526 V=800.0 PL=0
MOVL C01527 V=800.0 PL=0
MOVL C01528 V=800.0 PL=0
MOVL C01529 V=800.0 PL=0
MOVL C01530 V=800.0 PL=0
MOVL C01531 V=800.0 PL=0
MOVL C01532 V=800.0 PL=0
MOVL C01533 V=800.0 PL=0
MOVL C01534 V=800.0 PL=0
MOVL C01535 V=800.0 PL=0
MOVL C01536 V=800.0 PL=0
MOVL C01537 V=800.0 PL=0
MOVL C01538 V=800.0 PL=0
MOVL C01539 V=800.0 PL=0
MOVL C01540 V=800.0 PL=0
MOVL C01541 V=800.0 PL=0
MOVL C01542 V=800.0 PL=0
MOVL C01543 V=800.0 PL=0
MOVL C01544 V=800.0 PL=0
MOVL C01545 V=800.0 PL=0
MOVL C01546 V=800.0 PL=0
MOVL C01547 V=800.0 PL=0
MOVL C01548 V=800.0 PL=0
MOVL C01549 V=800.0 PL=0
MOVL C01550 V=800.0 PL=0
MOVL C01551 V=800.0 PL=0
MOVL C01552 V=800.0 PL=0
MOVL C01553 V=800.0 PL=0
MOVL C01554 V=800.0 PL=0
MOVL C01555 V=800.0 PL=0
MOVL C01556 V=800.0 PL=0
MOVL C01557 V=800.0 PL=0
MOVL C01558 V=800.0 PL=0
MOVL C01559 V=800.0 PL=0
MOVL C01560 V=800.0 PL=0
MOVL C01561 V=800.0 PL=0
MOVL C01562 V=800.0 PL=0
MOVL C01563 V=800.0 PL=0
MOVL C01564 V=800.0 PL=0
MOVL C01565 V=800.0 PL=0
MOVL C01566 V=800.0 PL=0
MOVL C01567 V=800.0 PL=0
MOVL C01568 V=800.0 PL=0
MOVL C01569 V=800.0 PL=0
MOVL C01570 V=800.0 PL=0
MOVL C01571 V=800.0 PL=0
MOVL C01572 V=800.0 PL=0
MOVL C01573 V=800.0 PL=0
MOVL C01574 V=800.0 PL=0
MOVL C01575 V=800.0 PL=0
MOVL C01576 V=800.0 PL=0
MOVL C01577 V=800.0 PL=0
MOVL C01578 V=800.0 PL=0
MOVL C01579 V=800.0 PL=0
MOVL C01580 V=800.0 PL=0
MOVL C01581 V=800.0 PL=0
MOVL C01582 V=800.0 PL=0
MOVL C01583 V=800.0 PL=0
MOVL C01584 V=800.0 PL=0
MOVL C01585 V=800.0 PL=0
MOVL C01586 V=800.0 PL=0
MOVL C01587 V=800.0 PL=0
MOVL C01588 V=800.0 PL=0
MOVL C01589 V=800.0 PL=0
MOVL C01590 V=800.0 PL=0
MOVL C01591 V=800.0 PL=0
MOVL C01592 V=800.0 PL=0
MOVL C01593 V=800.0 PL=0
MOVL C01594 V=800.0 PL=0
MOVL C01595 V=800.0 PL=0
MOVL C01596 V=800.0 PL=0
MOVL C01597 V=800.0 PL=0
MOVL C01598 V=800.0 PL=0
MOVL C01599 V=800.0 PL=0
MOVL C01600 V=800.0 PL=0
MOVL C01601 V=800.0 PL=0
MOVL C01602 V=800.0 PL=0
MOVL C01603 V=800.0 PL=0
MOVL C01604 V=800.0 PL=0
MOVL C01605 V=800.0 PL=0
MOVL C01606 V=800.0 PL=0
MOVL C01607 V=800.0 PL=0
MOVL C01608 V=800.0 PL=0
MOVL C01609 V=800.0 PL=0
MOVL C01610 V=800.0 PL=0
MOVL C01611 V=800.0 PL=0
MOVL C01612 V=800.0 PL=0
MOVL C01613 V=800.0 PL=0
MOVL C01614 V=800.0 PL=0
MOVL C01615 V=800.0 PL=0
MOVL C01616 V=800.0 PL=0
MOVL C01617 V=800.0 PL=0
MOVL C01618 V=800.0 PL=0
MOVL C01619 V=800.0 PL=0
MOVL C01620 V=800.0 PL=0
MOVL C01621 V=800.0 PL=0
MOVL C01622 V=800.0 PL=0
MOVL C01623 V=800.0 PL=0
MOVL C01624 V=800.0 PL=0
MOVL C01625 V=800.0 PL=0
MOVL C01626 V=800.0 PL=0
MOVL C01627 V=800.0 PL=0
MOVL C01628 V=800.0 PL=0
MOVL C01629 V=800.0 PL=0
MOVL C01630 V=800.0 PL=0
MOVL C01631 V=800.0 PL=0
MOVL C01632 V=800.0 PL=0
MOVL C01633 V=800.0 PL=0
MOVL C01634 V=800.0 PL=0
MOVL C01635 V=800.0 PL=0
MOVL C01636 V=800.0 PL=0
MOVL C01637 V=800.0 PL=0
MOVL C01638 V=800.0 PL=0
MOVL C01639 V=800.0 PL=0
MOVL C01640 V=800.0 PL=0
MOVL C01641 V=800.0 PL=0
MOVL C01642 V=800.0 PL=0
MOVL C01643 V=800.0 PL=0
MOVL C01644 V=800.0 PL=0
MOVL C01645 V=800.0 PL=0
MOVL C01646 V=800.0 PL=0
MOVL C01647 V=800.0 PL=0
MOVL C01648 V=800.0 PL=0
MOVL C01649 V=800.0 PL=0
MOVL C01650 V=800.0 PL=0
MOVL C01651 V=800.0 PL=0
MOVL C01652 V=800.0 PL=0
MOVL C01653 V=800.0 PL=0
MOVL C01654 V=800.0 PL=0
MOVL C01655 V=800.0 PL=0
MOVL C01656 V=800.0 PL=0
MOVL C01657 V=800.0 PL=0
MOVL C01658 V=800.0 PL=0
MOVL C01659 V=800.0 PL=0
MOVL C01660 V=800.0 PL=0
MOVL C01661 V=800.0 PL=0
MOVL C01662 V=800.0 PL=0
MOVL C01663 V=800.0 PL=0
MOVL C01664 V=800.0 PL=0
MOVL C01665 V=800.0 PL=0
MOVL C01666 V=800.0 PL=0
MOVL C01667 V=800.0 PL=0
MOVL C01668 V=800.0 PL=0
MOVL C01669 V=800.0 PL=0
MOVL C01670 V=800.0 PL=0
MOVL C01671 V=800.0 PL=0
MOVL C01672 V=800.0 PL=0
MOVL C01673 V=800.0 PL=0
MOVL C01674 V=800.0 PL=0
MOVL C01675 V=800.0 PL=0
MOVL C01676 V=800.0 PL=0
MOVL C01677 V=800.0 PL=0
MOVL C01678 V=800.0 PL=0
MOVL C01679 V=800.0 PL=0
MOVL C01680 V=800.0 PL=0
MOVL C01681 V=800.0 PL=0
MOVL C01682 V=800.0 PL=0
MOVL C01683 V=800.0 PL=0
MOVL C01684 V=800.0 PL=0
MOVL C01685 V=800.0 PL=0
MOVL C01686 V=800.0 PL=0
MOVL C01687 V=800.0 PL=0
MOVL C01688 V=800.0 PL=0
MOVL C01689 V=800.0 PL=0
MOVL C01690 V=800.0 PL=0
MOVL C01691 V=800.0 PL=0
MOVL C01692 V=800.0 PL=0
MOVL C01693 V=800.0 PL=0
MOVL C01694 V=800.0 PL=0
MOVL C01695 V=800.0 PL=0
MOVL C01696 V=800.0 PL=0
MOVL C01697 V=800.0 PL=0
MOVL C01698 V=800.0 PL=0
MOVL C01699 V=800.0 PL=0
MOVL C01700 V=800.0 PL=0
MOVL C01701 V=800.0 PL=0
MOVL C01702 V=800.0 PL=0
MOVL C01703 V=800.0 PL=0
MOVL C01704 V=800.0 PL=0
MOVL C01705 V=800.0 PL=0
MOVL C01706 V=800.0 PL=0
MOVL C01707 V=800.0 PL=0
MOVL C01708 V=800.0 PL=0
MOVL C01709 V=800.0 PL=0
MOVL C01710 V=800.0 PL=0
MOVL C01711 V=800.0 PL=0
MOVL C01712 V=800.0 PL=0
MOVL C01713 V=800.0 PL=0
MOVL C01714 V=800.0 PL=0
MOVL C01715 V=800.0 PL=0
MOVL C01716 V=800.0 PL=0
MOVL C01717 V=800.0 PL=0
MOVL C01718 V=800.0 PL=0
MOVL C01719 V=800.0 PL=0
MOVL C01720 V=800.0 PL=0
MOVL C01721 V=800.0 PL=0
MOVL C01722 V=800.0 PL=0
MOVL C01723 V=800.0 PL=0
MOVL C01724 V=800.0 PL=0
MOVL C01725 V=800.0 PL=0
MOVL C01726 V=800.0 PL=0
MOVL C01727 V=800.0 PL=0
MOVL C01728 V=800.0 PL=0
MOVL C01729 V=800.0 PL=0
MOVL C01730 V=800.0 PL=0
MOVL C01731 V=800.0 PL=0
MOVL C01732 V=800.0 PL=0
MOVL C01733 V=800.0 PL=0
MOVL C01734 V=800.0 PL=0
MOVL C01735 V=800.0 PL=0
MOVL C01736 V=800.0 PL=0
MOVL C01737 V=800.0 PL=0
MOVL C01738 V=800.0 PL=0
MOVL C01739 V=800.0 PL=0
MOVL C01740 V=800.0 PL=0
MOVL C01741 V=800.0 PL=0
MOVL C01742 V=800.0 PL=0
MOVL C01743 V=800.0 PL=0
MOVL C01744 V=800.0 PL=0
MOVL C01745 V=800.0 PL=0
MOVL C01746 V=800.0 PL=0
MOVL C01747 V=800.0 PL=0
MOVL C01748 V=800.0 PL=0
MOVL C01749 V=800.0 PL=0
MOVL C01750 V=800.0 PL=0
MOVL C01751 V=800.0 PL=0
MOVL C01752 V=800.0 PL=0
MOVL C01753 V=800.0 PL=0
MOVL C01754 V=800.0 PL=0
MOVL C01755 V=800.0 PL=0
MOVL C01756 V=800.0 PL=0
MOVL C01757 V=800.0 PL=0
MOVL C01758 V=800.0 PL=0
MOVL C01759 V=800.0 PL=0
MOVL C01760 V=800.0 PL=0
MOVL C01761 V=800.0 PL=0
MOVL C01762 V=800.0 PL=0
MOVL C01763 V=800.0 PL=0
MOVL C01764 V=800.0 PL=0
MOVL C01765 V=800.0 PL=0
MOVL C01766 V=800.0 PL=0
MOVL C01767 V=800.0 PL=0
MOVL C01768 V=800.0 PL=0
MOVL C01769 V=800.0 PL=0
MOVL C01770 V=800.0 PL=0
MOVL C01771 V=800.0 PL=0
MOVL C01772 V=800.0 PL=0
MOVL C01773 V=800.0 PL=0
MOVL C01774 V=800.0 PL=0
MOVL C01775 V=800.0 PL=0
MOVL C01776 V=800.0 PL=0
MOVL C01777 V=800.0 PL=0
MOVL C01778 V=800.0 PL=0
MOVL C01779 V=800.0 PL=0
MOVL C01780 V=800.0 PL=0
MOVL C01781 V=800.0 PL=0
MOVL C01782 V=800.0 PL=0
MOVL C01783 V=800.0 PL=0
MOVL C01784 V=800.0 PL=0
MOVL C01785 V=800.0 PL=0
MOVL C01786 V=800.0 PL=0
MOVL C01787 V=800.0 PL=0
MOVL C01788 V=800.0 PL=0
MOVL C01789 V=800.0 PL=0
MOVL C01790 V=800.0 PL=0
MOVL C01791 V=800.0 PL=0
MOVL C01792 V=800.0 PL=0
MOVL C01793 V=800.0 PL=0
MOVL C01794 V=800.0 PL=0
MOVL C01795 V=800.0 PL=0
MOVL C01796 V=800.0 PL=0
MOVL C01797 V=800.0 PL=0
MOVL C01798 V=800.0 PL=0
MOVL C01799 V=800.0 PL=0
MOVL C01800 V=800.0 PL=0
MOVL C01801 V=800.0 PL=0
MOVL C01802 V=800.0 PL=0
MOVL C01803 V=800.0 PL=0
MOVL C01804 V=800.0 PL=0
MOVL C01805 V=800.0 PL=0
MOVL C01806 V=800.0 PL=0
MOVL C01807 V=800.0 PL=0
MOVL C01808 V=800.0 PL=0
MOVL C01809 V=800.0 PL=0
MOVL C01810 V=800.0 PL=0
MOVL C01811 V=800.0 PL=0
MOVL C01812 V=800.0 PL=0
MOVL C01813 V=800.0 PL=0
MOVL C01814 V=800.0 PL=0
MOVL C01815 V=800.0 PL=0
MOVL C01816 V=800.0 PL=0
MOVL C01817 V=800.0 PL=0
MOVL C01818 V=800.0 PL=0
MOVL C01819 V=800.0 PL=0
MOVL C01820 V=800.0 PL=0
MOVL C01821 V=800.0 PL=0
MOVL C01822 V=800.0 PL=0
MOVL C01823 V=800.0 PL=0
MOVL C01824 V=800.0 PL=0
MOVL C01825 V=800.0 PL=0
MOVL C01826 V=800.0 PL=0
MOVL C01827 V=800.0 PL=0
MOVL C01828 V=800.0 PL=0
MOVL C01829 V=800.0 PL=0
MOVL C01830 V=800.0 PL=0
MOVL C01831 V=800.0 PL=0
MOVL C01832 V=800.0 PL=0
MOVL C01833 V=800.0 PL=0
MOVL C01834 V=800.0 PL=0
MOVL C01835 V=800.0 PL=0
MOVL C01836 V=800.0 PL=0
MOVL C01837 V=800.0 PL=0
MOVL C01838 V=800.0 PL=0
MOVL C01839 V=800.0 PL=0
MOVL C01840 V=800.0 PL=0
MOVL C01841 V=800.0 PL=0
MOVL C01842 V=800.0 PL=0
MOVL C01843 V=800.0 PL=0
MOVL C01844 V=800.0 PL=0
MOVL C01845 V=800.0 PL=0
MOVL C01846 V=800.0 PL=0
MOVL C01847 V=800.0 PL=0
MOVL C01848 V=800.0 PL=0
MOVL C01849 V=800.0 PL=0
MOVL C01850 V=800.0 PL=0
MOVL C01851 V=800.0 PL=0
MOVL C01852 V=800.0 PL=0
MOVL C01853 V=800.0 PL=0
MOVL C01854 V=800.0 PL=0
MOVL C01855 V=800.0 PL=0
MOVL C01856 V=800.0 PL=0
MOVL C01857 V=800.0 PL=0
MOVL C01858 V=800.0 PL=0
MOVL C01859 V=800.0 PL=0
MOVL C01860 V=800.0 PL=0
MOVL C01861 V=800.0 PL=0
MOVL C01862 V=800.0 PL=0
MOVL C01863 V=800.0 PL=0
MOVL C01864 V=800.0 PL=0
MOVL C01865 V=800.0 PL=0
MOVL C01866 V=800.0 PL=0
MOVL C01867 V=800.0 PL=0
MOVL C01868 V=800.0 PL=0
MOVL C01869 V=800.0 PL=0
MOVL C01870 V=800.0 PL=0
MOVL C01871 V=800.0 PL=0
MOVL C01872 V=800.0 PL=0
MOVL C01873 V=800.0 PL=0
MOVL C01874 V=800.0 PL=0
MOVL C01875 V=800.0 PL=0
MOVL C01876 V=800.0 PL=0
MOVL C01877 V=800.0 PL=0
MOVL C01878 V=800.0 PL=0
MOVL C01879 V=800.0 PL=0
MOVL C01880 V=800.0 PL=0
MOVL C01881 V=800.0 PL=0
MOVL C01882 V=800.0 PL=0
MOVL C01883 V=800.0 PL=0
MOVL C01884 V=800.0 PL=0
MOVL C01885 V=800.0 PL=0
MOVL C01886 V=800.0 PL=0
MOVL C01887 V=800.0 PL=0
MOVL C01888 V=800.0 PL=0
MOVL C01889 V=800.0 PL=0
MOVL C01890 V=800.0 PL=0
MOVL C01891 V=800.0 PL=0
MOVL C01892 V=800.0 PL=0
MOVL C01893 V=800.0 PL=0
MOVL C01894 V=800.0 PL=0
MOVL C01895 V=800.0 PL=0
MOVL C01896 V=800.0 PL=0
MOVL C01897 V=800.0 PL=0
MOVL C01898 V=800.0 PL=0
MOVL C01899 V=800.0 PL=0
MOVL C01900 V=800.0 PL=0
MOVL C01901 V=800.0 PL=0
MOVL C01902 V=800.0 PL=0
MOVL C01903 V=800.0 PL=0
MOVL C01904 V=800.0 PL=0
MOVL C01905 V=800.0 PL=0
MOVL C01906 V=800.0 PL=0
MOVL C01907 V=800.0 PL=0
MOVL C01908 V=800.0 PL=0
MOVL C01909 V=800.0 PL=0
MOVL C01910 V=800.0 PL=0
MOVL C01911 V=800.0 PL=0
MOVL C01912 V=800.0 PL=0
MOVL C01913 V=800.0 PL=0
MOVL C01914 V=800.0 PL=0
MOVL C01915 V=800.0 PL=0
MOVL C01916 V=800.0 PL=0
MOVL C01917 V=800.0 PL=0
MOVL C01918 V=800.0 PL=0
MOVL C01919 V=800.0 PL=0
MOVL C01920 V=800.0 PL=0
MOVL C01921 V=800.0 PL=0
MOVL C01922 V=800.0 PL=0
MOVL C01923 V=800.0 PL=0
MOVL C01924 V=800.0 PL=0
MOVL C01925 V=800.0 PL=0
MOVL C01926 V=800.0 PL=0
MOVL C01927 V=800.0 PL=0
MOVL C01928 V=800.0 PL=0
MOVL C01929 V=800.0 PL=0
MOVL C01930 V=800.0 PL=0
MOVL C01931 V=800.0 PL=0
MOVL C01932 V=800.0 PL=0
MOVL C01933 V=800.0 PL=0
MOVL C01934 V=800.0 PL=0
MOVL C01935 V=800.0 PL=0
MOVL C01936 V=800.0 PL=0
MOVL C01937 V=800.0 PL=0
MOVL C01938 V=800.0 PL=0
MOVL C01939 V=800.0 PL=0
MOVL C01940 V=800.0 PL=0
MOVL C01941 V=800.0 PL=0
MOVL C01942 V=800.0 PL=0
MOVL C01943 V=800.0 PL=0
MOVL C01944 V=800.0 PL=0
MOVL C01945 V=800.0 PL=0
MOVL C01946 V=800.0 PL=0
MOVL C01947 V=800.0 PL=0
MOVL C01948 V=800.0 PL=0
MOVL C01949 V=800.0 PL=0
MOVL C01950 V=800.0 PL=0
MOVL C01951 V=800.0 PL=0
MOVL C01952 V=800.0 PL=0
MOVL C01953 V=800.0 PL=0
MOVL C01954 V=800.0 PL=0
MOVL C01955 V=800.0 PL=0
MOVL C01956 V=800.0 PL=0
MOVL C01957 V=800.0 PL=0
MOVL C01958 V=800.0 PL=0
MOVL C01959 V=800.0 PL=0
MOVL C01960 V=800.0 PL=0
MOVL C01961 V=800.0 PL=0
MOVL C01962 V=800.0 PL=0
MOVL C01963 V=800.0 PL=0
MOVL C01964 V=800.0 PL=0
MOVL C01965 V=800.0 PL=0
MOVL C01966 V=800.0 PL=0
MOVL C01967 V=800.0 PL=0
MOVL C01968 V=800.0 PL=0
MOVL C01969 V=800.0 PL=0
